LIN {X 0,Y 517.926,Z 485.108,A -85,B 0,C 180,E1 -5117.361,E2 -5117.361} C_VEL
LIN {X 0,Y 517.662,Z 497.086,A -85,B 0,C 180,E1 -5118.063,E2 -5118.063} C_VEL
LIN {X 0,Y 517.369,Z 508.755,A -85,B 0,C 180,E1 -5118.938,E2 -5118.938} C_VEL
LIN {X 0,Y 517.043,Z 518.274,A -85,B 0,C 180,E1 -5119.822,E2 -5119.822} C_VEL
LIN {X 0,Y 516.815,Z 526.96,A -85,B 0,C 180,E1 -5120.806,E2 -5120.806} C_VEL
LIN {X 0,Y 516.617,Z 535.392,A -85,B 0,C 180,E1 -5121.985,E2 -5121.985} C_VEL
LIN {X 0,Y 516.477,Z 542.404,A -85,B 0,C 180,E1 -5123.204,E2 -5123.204} C_VEL
LIN {X 0,Y 516.405,Z 548.407,A -85,B 0,C 180,E1 -5124.533,E2 -5124.533} C_VEL
LIN {X 0,Y 516.343,Z 552.44,A -85,B 0,C 180,E1 -5125.707,E2 -5125.707} C_VEL
LIN {X 0,Y 516.282,Z 555.413,A -85,B 0,C 180,E1 -5126.879,E2 -5126.879} C_VEL
LIN {X 0,Y 516.261,Z 556.832,A -85,B 0,C 180,E1 -5127.659,E2 -5127.659} C_VEL
LIN {X 0,Y 516.16,Z 558.451,A -85,B 0,C 180,E1 -5129.22,E2 -5129.22} C_VEL
LIN {X 0,Y 516.155,Z 558.67,A -85,B 0,C 180,E1 -5130,E2 -5130} C_VEL
LIN {X 0,Y 516.16,Z 558.45,A -85,B 0,C 180,E1 -5130.78,E2 -5130.78} C_VEL
LIN {X 0,Y 516.261,Z 556.828,A -85,B 0,C 180,E1 -5132.341,E2 -5132.341} C_VEL
LIN {X 0,Y 516.282,Z 555.406,A -85,B 0,C 180,E1 -5133.121,E2 -5133.121} C_VEL
LIN {X 0,Y 516.343,Z 552.421,A -85,B 0,C 180,E1 -5134.293,E2 -5134.293} C_VEL
LIN {X 0,Y 516.405,Z 548.374,A -85,B 0,C 180,E1 -5135.467,E2 -5135.467} C_VEL
LIN {X 0,Y 516.465,Z 542.972,A -85,B 0,C 180,E1 -5136.679,E2 -5136.679} C_VEL
LIN {X 0,Y 516.579,Z 536.576,A -85,B 0,C 180,E1 -5137.819,E2 -5137.819} C_VEL
LIN {X 0,Y 516.771,Z 528.376,A -85,B 0,C 180,E1 -5138.998,E2 -5138.998} C_VEL
LIN {X 0,Y 516.993,Z 520.003,A -85,B 0,C 180,E1 -5139.981,E2 -5139.981} C_VEL
LIN {X 0,Y 517.292,Z 509.755,A -85,B 0,C 180,E1 -5140.965,E2 -5140.965} C_VEL
LIN {X 0,Y 517.549,Z 499.569,A -85,B 0,C 180,E1 -5141.753,E2 -5141.753} C_VEL
LIN {X 0,Y 517.84,Z 487.976,A -85,B 0,C 180,E1 -5142.47,E2 -5142.47} C_VEL
LIN {X 0,Y 518.063,Z 476.175,A -85,B 0,C 180,E1 -5143.034,E2 -5143.034} C_VEL
LIN {X 0,Y 518.291,Z 463.332,A -85,B 0,C 180,E1 -5143.478,E2 -5143.478} C_VEL
LIN {X 0,Y 518.127,Z 456.266,A -85,B 0,C 180,E1 -5143.657,E2 -5143.657} C_VEL
LIN {X 0,Y 516.991,Z 447.207,A -85,B 0,C 180,E1 -5143.863,E2 -5143.863} C_VEL
LIN {X 0,Y 517.273,Z 430.127,A -85,B 0,C 180,E1 -5146.781,E2 -5146.781} C_VEL
LIN {X 0,Y 517.596,Z 415.01,A -85,B 0,C 180,E1 -5149.431,E2 -5149.431} C_VEL
LIN {X 0,Y 517.925,Z 402.35,A -85,B 0,C 180,E1 -5151.702,E2 -5151.702} C_VEL
LIN {X 0,Y 518.488,Z 388.132,A -85,B 0,C 180,E1 -5154.383,E2 -5154.383} C_VEL
LIN {X 0,Y 519.352,Z 373.06,A -85,B 0,C 180,E1 -5157.394,E2 -5157.394} C_VEL
LIN {X 0,Y 519.545,Z 368.168,A -85,B 0,C 180,E1 -5158.445,E2 -5158.445} C_VEL
LIN {X 0,Y 517.68,Z 359.516,A -85,B 0,C 180,E1 -5160.604,E2 -5160.604} C_VEL
LIN {X 0,Y 516.886,Z 356.103,A -85,B 0,C 180,E1 -5161.566,E2 -5161.566} C_VEL
LIN {X 0,Y 516.911,Z 356.099,A -85,B 0,C 180,E1 -5163.966,E2 -5163.966} C_VEL
LIN {X 0,Y 516.879,Z 356.103,A -85,B 0,C 180,E1 -5166.746,E2 -5166.746} C_VEL
LIN {X 0,Y 516.885,Z 356.102,A -85,B 0,C 180,E1 -5169.721,E2 -5169.721} C_VEL
LIN {X 0,Y 516.91,Z 356.1,A -85,B 0,C 180,E1 -5172.761,E2 -5172.761} C_VEL
LIN {X 0,Y 516.926,Z 356.097,A -85,B 0,C 180,E1 -5175.01,E2 -5175.01} C_VEL
LIN {X 0,Y 516.921,Z 356.097,A -85,B 0,C 180,E1 -5178.398,E2 -5178.398} C_VEL
LIN {X 0,Y 516.91,Z 356.1,A -85,B 0,C 180,E1 -5181.287,E2 -5181.287} C_VEL
LIN {X 0,Y 516.89,Z 356.103,A -85,B 0,C 180,E1 -5184.221,E2 -5184.221} C_VEL
LIN {X 0,Y 516.9,Z 356.102,A -85,B 0,C 180,E1 -5187.053,E2 -5187.053} C_VEL
LIN {X 0,Y 516.926,Z 356.236,A -85,B 0,C 180,E1 -5189.153,E2 -5189.153} C_VEL
LIN {X 0,Y 517.195,Z 359.452,A -85,B 0,C 180,E1 -5190.712,E2 -5190.712} C_VEL
LIN {X 0,Y 517.047,Z 365.951,A -85,B 0,C 180,E1 -5193.781,E2 -5193.781} C_VEL
LIN {X 0,Y 516.896,Z 372.331,A -85,B 0,C 180,E1 -5196.778,E2 -5196.778} C_VEL
LIN {X 0,Y 516.762,Z 378.758,A -85,B 0,C 180,E1 -5199.786,E2 -5199.786} C_VEL
LIN {X 0,Y 516.703,Z 384.815,A -85,B 0,C 180,E1 -5202.588,E2 -5202.588} C_VEL
LIN {X 0,Y 516.634,Z 390.136,A -85,B 0,C 180,E1 -5205.021,E2 -5205.021} C_VEL
LIN {X 0,Y 516.491,Z 397.626,A -85,B 0,C 180,E1 -5208.442,E2 -5208.442} C_VEL
LIN {X 0,Y 516.412,Z 405.171,A -85,B 0,C 180,E1 -5211.809,E2 -5211.809} C_VEL
LIN {X 0,Y 517.193,Z 411.851,A -85,B 0,C 180,E1 -5212.092,E2 -5212.092} C_VEL
LIN {X 0,Y 517.076,Z 421.865,A -85,B 0,C 180,E1 -5212.62,E2 -5212.62} C_VEL
LIN {X 0,Y 516.967,Z 430.533,A -85,B 0,C 180,E1 -5213.252,E2 -5213.252} C_VEL
LIN {X 0,Y 516.779,Z 437.867,A -85,B 0,C 180,E1 -5213.95,E2 -5213.95} C_VEL
LIN {X 0,Y 516.671,Z 444.225,A -85,B 0,C 180,E1 -5214.732,E2 -5214.732} C_VEL
LIN {X 0,Y 516.564,Z 449.253,A -85,B 0,C 180,E1 -5215.513,E2 -5215.513} C_VEL
LIN {X 0,Y 516.546,Z 454.014,A -85,B 0,C 180,E1 -5216.49,E2 -5216.49} C_VEL
LIN {X 0,Y 516.333,Z 457.969,A -85,B 0,C 180,E1 -5217.66,E2 -5217.66} C_VEL
LIN {X 0,Y 516.266,Z 459.663,A -85,B 0,C 180,E1 -5218.44,E2 -5218.44} C_VEL
LIN {X 0,Y 516.246,Z 460.666,A -85,B 0,C 180,E1 -5219.22,E2 -5219.22} C_VEL
LIN {X 0,Y 516.24,Z 461.005,A -85,B 0,C 180,E1 -5220,E2 -5220} C_VEL
LIN {X 0,Y 516.239,Z 460.689,A -85,B 0,C 180,E1 -5220.78,E2 -5220.78} C_VEL
LIN {X 0,Y 516.255,Z 459.71,A -85,B 0,C 180,E1 -5221.56,E2 -5221.56} C_VEL
LIN {X 0,Y 516.421,Z 456.909,A -85,B 0,C 180,E1 -5222.73,E2 -5222.73} C_VEL
LIN {X 0,Y 516.543,Z 454.125,A -85,B 0,C 180,E1 -5223.51,E2 -5223.51} C_VEL
LIN {X 0,Y 516.558,Z 449.409,A -85,B 0,C 180,E1 -5224.487,E2 -5224.487} C_VEL
LIN {X 0,Y 516.634,Z 444.423,A -85,B 0,C 180,E1 -5225.269,E2 -5225.269} C_VEL
LIN {X 0,Y 516.662,Z 438.145,A -85,B 0,C 180,E1 -5226.052,E2 -5226.052} C_VEL
LIN {X 0,Y 516.878,Z 430.436,A -85,B 0,C 180,E1 -5226.788,E2 -5226.788} C_VEL
LIN {X 0,Y 516.993,Z 421.754,A -85,B 0,C 180,E1 -5227.42,E2 -5227.42} C_VEL
LIN {X 0,Y 517.128,Z 411.453,A -85,B 0,C 180,E1 -5227.958,E2 -5227.958} C_VEL
LIN {X 0,Y 516.329,Z 404.462,A -85,B 0,C 180,E1 -5228.242,E2 -5228.242} C_VEL
LIN {X 0,Y 516.353,Z 396.845,A -85,B 0,C 180,E1 -5231.483,E2 -5231.483} C_VEL
LIN {X 0,Y 516.469,Z 389.182,A -85,B 0,C 180,E1 -5234.949,E2 -5234.949} C_VEL
LIN {X 0,Y 516.579,Z 382.087,A -85,B 0,C 180,E1 -5238.235,E2 -5238.235} C_VEL
LIN {X 0,Y 516.645,Z 376.784,A -85,B 0,C 180,E1 -5240.713,E2 -5240.713} C_VEL
LIN {X 0,Y 516.693,Z 371.107,A -85,B 0,C 180,E1 -5243.232,E2 -5243.232} C_VEL
LIN {X 0,Y 516.825,Z 364.647,A -85,B 0,C 180,E1 -5246.169,E2 -5246.169} C_VEL
LIN {X 0,Y 516.974,Z 357.423,A -85,B 0,C 180,E1 -5249.535,E2 -5249.535} C_VEL
LIN {X 0,Y 517.006,Z 356.086,A -85,B 0,C 180,E1 -5250.197,E2 -5250.197} C_VEL
LIN {X 0,Y 516.915,Z 356.093,A -85,B 0,C 180,E1 -5253.879,E2 -5253.879} C_VEL
LIN {X 0,Y 516.886,Z 356.099,A -85,B 0,C 180,E1 -5256.746,E2 -5256.746} C_VEL
LIN {X 0,Y 516.886,Z 356.101,A -85,B 0,C 180,E1 -5259.721,E2 -5259.721} C_VEL
LIN {X 0,Y 516.917,Z 356.095,A -85,B 0,C 180,E1 -5261.775,E2 -5261.775} C_VEL
LIN {X 0,Y 516.927,Z 356.094,A -85,B 0,C 180,E1 -5265.01,E2 -5265.01} C_VEL
LIN {X 0,Y 516.92,Z 356.095,A -85,B 0,C 180,E1 -5268.398,E2 -5268.398} C_VEL
LIN {X 0,Y 516.886,Z 356.101,A -85,B 0,C 180,E1 -5269.481,E2 -5269.481} C_VEL
LIN {X 0,Y 516.226,Z 356.185,A -85,B 0,C 180,E1 -5270.132,E2 -5270.132} C_VEL
LIN {X 0,Y 513.357,Z 356.543,A -85,B 0,C 180,E1 -5271.189,E2 -5271.189} C_VEL
LIN {X 0,Y 510.931,Z 356.843,A -85,B 0,C 180,E1 -5272.04,E2 -5272.04} C_VEL
LIN {X 0,Y 509.898,Z 356.972,A -85,B 0,C 180,E1 -5272.697,E2 -5272.697} C_VEL
LIN {X 0,Y 509.818,Z 356.981,A -85,B 0,C 180,E1 -5272.92,E2 -5272.92} C_VEL
LIN {X 0,Y 509.86,Z 356.973,A -85,B 0,C 180,E1 -5275.797,E2 -5275.797} C_VEL
LIN {X 0,Y 509.85,Z 356.975,A -85,B 0,C 180,E1 -5278.72,E2 -5278.72} C_VEL
LIN {X 0,Y 509.902,Z 356.969,A -85,B 0,C 180,E1 -5281.899,E2 -5281.899} C_VEL
LIN {X 0,Y 509.845,Z 356.979,A -85,B 0,C 180,E1 -5284.702,E2 -5284.702} C_VEL
LIN {X 0,Y 509.831,Z 356.977,A -85,B 0,C 180,E1 -5287.458,E2 -5287.458} C_VEL
LIN {X 0,Y 509.921,Z 356.97,A -85,B 0,C 180,E1 -5289.845,E2 -5289.845} C_VEL
LIN {X 0,Y 509.886,Z 356.973,A -85,B 0,C 180,E1 -5293.175,E2 -5293.175} C_VEL
LIN {X 0,Y 509.868,Z 356.972,A -85,B 0,C 180,E1 -5295.634,E2 -5295.634} C_VEL
LIN {X 0,Y 509.918,Z 356.966,A -85,B 0,C 180,E1 -5298.875,E2 -5298.875} C_VEL
LIN {X 0,Y 509.956,Z 356.962,A -85,B 0,C 180,E1 -5302.078,E2 -5302.078} C_VEL
LIN {X 0,Y 509.985,Z 356.962,A -85,B 0,C 180,E1 -5304.464,E2 -5304.464} C_VEL
LIN {X 0,Y 510.059,Z 356.949,A -85,B 0,C 180,E1 -5307.631,E2 -5307.631} C_VEL
LIN {X 0,Y 510.068,Z 356.948,A -85,B 0,C 180,E1 -5310.789,E2 -5310.789} C_VEL
LIN {X 0,Y 509.958,Z 356.965,A -85,B 0,C 180,E1 -5313.16,E2 -5313.16} C_VEL
LIN {X 0,Y 509.958,Z 356.965,A -85,B 0,C 180,E1 -5316.33,E2 -5316.33} C_VEL
LIN {X 0,Y 509.919,Z 356.964,A -85,B 0,C 180,E1 -5318.72,E2 -5318.72} C_VEL
LIN {X 0,Y 509.909,Z 356.968,A -85,B 0,C 180,E1 -5321.932,E2 -5321.932} C_VEL
LIN {X 0,Y 509.898,Z 356.969,A -85,B 0,C 180,E1 -5325.242,E2 -5325.242} C_VEL
LIN {X 0,Y 509.893,Z 356.974,A -85,B 0,C 180,E1 -5328.001,E2 -5328.001} C_VEL
LIN {X 0,Y 509.854,Z 356.975,A -85,B 0,C 180,E1 -5331.002,E2 -5331.002} C_VEL
LIN {X 0,Y 509.869,Z 356.975,A -85,B 0,C 180,E1 -5334.426,E2 -5334.426} C_VEL
LIN {X 0,Y 509.889,Z 356.97,A -85,B 0,C 180,E1 -5337.055,E2 -5337.055} C_VEL
LIN {X 0,Y 509.861,Z 356.977,A -85,B 0,C 180,E1 -5339.751,E2 -5339.751} C_VEL
LIN {X 0,Y 509.878,Z 356.973,A -85,B 0,C 180,E1 -5342.774,E2 -5342.774} C_VEL
LIN {X 0,Y 509.829,Z 356.977,A -85,B 0,C 180,E1 -5345.578,E2 -5345.578} C_VEL
LIN {X 0,Y 509.854,Z 356.977,A -85,B 0,C 180,E1 -5348.338,E2 -5348.338} C_VEL
LIN {X 0,Y 509.858,Z 356.978,A -85,B 0,C 180,E1 -5351.425,E2 -5351.425} C_VEL
LIN {X 0,Y 509.86,Z 356.977,A -85,B 0,C 180,E1 -5354.668,E2 -5354.668} C_VEL
LIN {X 0,Y 509.858,Z 356.977,A -85,B 0,C 180,E1 -5358.103,E2 -5358.103} C_VEL
LIN {X 0,Y 509.849,Z 356.974,A -85,B 0,C 180,E1 -5360.647,E2 -5360.647} C_VEL
LIN {X 0,Y 509.827,Z 356.977,A -85,B 0,C 180,E1 -5363.647,E2 -5363.647} C_VEL
LIN {X 0,Y 509.862,Z 356.978,A -85,B 0,C 180,E1 -5366.539,E2 -5366.539} C_VEL
LIN {X 0,Y 509.848,Z 356.977,A -85,B 0,C 180,E1 -5369.334,E2 -5369.334} C_VEL
LIN {X 0,Y 509.895,Z 356.968,A -85,B 0,C 180,E1 -5372.054,E2 -5372.054} C_VEL
LIN {X 0,Y 509.88,Z 356.975,A -85,B 0,C 180,E1 -5374.704,E2 -5374.704} C_VEL
LIN {X 0,Y 509.84,Z 356.976,A -85,B 0,C 180,E1 -5377.455,E2 -5377.455} C_VEL
LIN {X 0,Y 509.92,Z 356.969,A -85,B 0,C 180,E1 -5379.845,E2 -5379.845} C_VEL
LIN {X 0,Y 509.887,Z 356.973,A -85,B 0,C 180,E1 -5383.175,E2 -5383.175} C_VEL
LIN {X 0,Y 509.867,Z 356.971,A -85,B 0,C 180,E1 -5385.634,E2 -5385.634} C_VEL
LIN {X 0,Y 509.925,Z 356.965,A -85,B 0,C 180,E1 -5388.875,E2 -5388.875} C_VEL
LIN {X 0,Y 509.955,Z 356.962,A -85,B 0,C 180,E1 -5392.078,E2 -5392.078} C_VEL
LIN {X 0,Y 509.985,Z 356.96,A -85,B 0,C 180,E1 -5394.464,E2 -5394.464} C_VEL
LIN {X 0,Y 510.058,Z 356.949,A -85,B 0,C 180,E1 -5397.631,E2 -5397.631} C_VEL
LIN {X 0,Y 510.067,Z 356.948,A -85,B 0,C 180,E1 -5400.789,E2 -5400.789} C_VEL
LIN {X 0,Y 509.96,Z 356.964,A -85,B 0,C 180,E1 -5403.16,E2 -5403.16} C_VEL
LIN {X 0,Y 509.981,Z 356.962,A -85,B 0,C 180,E1 -5406.33,E2 -5406.33} C_VEL
LIN {X 0,Y 509.915,Z 356.967,A -85,B 0,C 180,E1 -5408.72,E2 -5408.72} C_VEL
LIN {X 0,Y 509.907,Z 356.969,A -85,B 0,C 180,E1 -5411.932,E2 -5411.932} C_VEL
LIN {X 0,Y 509.897,Z 356.97,A -85,B 0,C 180,E1 -5415.242,E2 -5415.242} C_VEL
LIN {X 0,Y 509.869,Z 356.975,A -85,B 0,C 180,E1 -5417.993,E2 -5417.993} C_VEL
LIN {X 0,Y 509.889,Z 356.97,A -85,B 0,C 180,E1 -5420.402,E2 -5420.402} C_VEL
LIN {X 0,Y 509.832,Z 356.979,A -85,B 0,C 180,E1 -5423.563,E2 -5423.563} C_VEL
LIN {X 0,Y 509.914,Z 356.972,A -85,B 0,C 180,E1 -5426.378,E2 -5426.378} C_VEL
LIN {X 0,Y 509.879,Z 356.969,A -85,B 0,C 180,E1 -5428.844,E2 -5428.844} C_VEL
LIN {X 0,Y 509.823,Z 356.983,A -85,B 0,C 180,E1 -5431.59,E2 -5431.59} C_VEL
LIN {X 0,Y 509.855,Z 356.976,A -85,B 0,C 180,E1 -5434.413,E2 -5434.413} C_VEL
LIN {X 0,Y 509.822,Z 356.978,A -85,B 0,C 180,E1 -5437.34,E2 -5437.34} C_VEL
LIN {X 0,Y 509.84,Z 356.975,A -85,B 0,C 180,E1 -5440.382,E2 -5440.382} C_VEL
LIN {X 0,Y 509.842,Z 356.979,A -85,B 0,C 180,E1 -5443.064,E2 -5443.064} C_VEL
LIN {X 0,Y 509.833,Z 356.977,A -85,B 0,C 180,E1 -5445.792,E2 -5445.792} C_VEL
LIN {X 0,Y 509.86,Z 356.974,A -85,B 0,C 180,E1 -5448.575,E2 -5448.575} C_VEL
LIN {X 0,Y 509.853,Z 356.976,A -85,B 0,C 180,E1 -5451.787,E2 -5451.787} C_VEL
LIN {X 0,Y 509.832,Z 356.981,A -85,B 0,C 180,E1 -5454.622,E2 -5454.622} C_VEL
LIN {X 0,Y 509.866,Z 356.97,A -85,B 0,C 180,E1 -5457.481,E2 -5457.481} C_VEL
LIN {X 0,Y 509.875,Z 357.124,A -85,B 0,C 180,E1 -5458.865,E2 -5458.865} C_VEL
LIN {X 0,Y 512.351,Z 368.579,A -85,B 0,C 180,E1 -5461.39,E2 -5461.39} C_VEL
LIN {X 0,Y 512.386,Z 374.915,A -85,B 0,C 180,E1 -5462.646,E2 -5462.646} C_VEL
LIN {X 0,Y 511.54,Z 391.643,A -85,B 0,C 180,E1 -5465.875,E2 -5465.875} C_VEL
LIN {X 0,Y 510.912,Z 408.335,A -85,B 0,C 180,E1 -5469.044,E2 -5469.044} C_VEL
LIN {X 0,Y 510.492,Z 420.904,A -85,B 0,C 180,E1 -5471.332,E2 -5471.332} C_VEL
LIN {X 0,Y 510.154,Z 437.346,A -85,B 0,C 180,E1 -5474.204,E2 -5474.204} C_VEL
LIN {X 0,Y 509.97,Z 447.553,A -85,B 0,C 180,E1 -5475.994,E2 -5475.994} C_VEL
LIN {X 0,Y 511.367,Z 459.455,A -85,B 0,C 180,E1 -5476.261,E2 -5476.261} C_VEL
LIN {X 0,Y 511.148,Z 472.764,A -85,B 0,C 180,E1 -5476.685,E2 -5476.685} C_VEL
LIN {X 0,Y 510.938,Z 483.958,A -85,B 0,C 180,E1 -5477.185,E2 -5477.185} C_VEL
LIN {X 0,Y 510.66,Z 495.859,A -85,B 0,C 180,E1 -5477.878,E2 -5477.878} C_VEL
LIN {X 0,Y 510.293,Z 507.862,A -85,B 0,C 180,E1 -5478.782,E2 -5478.782} C_VEL
LIN {X 0,Y 510.011,Z 517.448,A -85,B 0,C 180,E1 -5479.68,E2 -5479.68} C_VEL
LIN {X 0,Y 509.759,Z 526.189,A -85,B 0,C 180,E1 -5480.677,E2 -5480.677} C_VEL
LIN {X 0,Y 509.538,Z 534.661,A -85,B 0,C 180,E1 -5481.872,E2 -5481.872} C_VEL
LIN {X 0,Y 509.401,Z 541.938,A -85,B 0,C 180,E1 -5483.156,E2 -5483.156} C_VEL
LIN {X 0,Y 509.344,Z 547.728,A -85,B 0,C 180,E1 -5484.457,E2 -5484.457} C_VEL
LIN {X 0,Y 509.268,Z 551.771,A -85,B 0,C 180,E1 -5485.647,E2 -5485.647} C_VEL
LIN {X 0,Y 509.232,Z 554.754,A -85,B 0,C 180,E1 -5486.835,E2 -5486.835} C_VEL
LIN {X 0,Y 509.19,Z 556.176,A -85,B 0,C 180,E1 -5487.627,E2 -5487.627} C_VEL
LIN {X 0,Y 509.09,Z 557.796,A -85,B 0,C 180,E1 -5489.209,E2 -5489.209} C_VEL
LIN {X 0,Y 509.086,Z 558.01,A -85,B 0,C 180,E1 -5490,E2 -5490} C_VEL
LIN {X 0,Y 509.09,Z 557.787,A -85,B 0,C 180,E1 -5490.791,E2 -5490.791} C_VEL
LIN {X 0,Y 509.19,Z 556.154,A -85,B 0,C 180,E1 -5492.373,E2 -5492.373} C_VEL
LIN {X 0,Y 509.232,Z 554.722,A -85,B 0,C 180,E1 -5493.165,E2 -5493.165} C_VEL
LIN {X 0,Y 509.268,Z 551.718,A -85,B 0,C 180,E1 -5494.353,E2 -5494.353} C_VEL
LIN {X 0,Y 509.344,Z 547.65,A -85,B 0,C 180,E1 -5495.543,E2 -5495.543} C_VEL
LIN {X 0,Y 509.402,Z 541.835,A -85,B 0,C 180,E1 -5496.844,E2 -5496.844} C_VEL
LIN {X 0,Y 509.563,Z 534.524,A -85,B 0,C 180,E1 -5498.127,E2 -5498.127} C_VEL
LIN {X 0,Y 509.759,Z 526.001,A -85,B 0,C 180,E1 -5499.323,E2 -5499.323} C_VEL
LIN {X 0,Y 510.006,Z 517.207,A -85,B 0,C 180,E1 -5500.32,E2 -5500.32} C_VEL
LIN {X 0,Y 510.33,Z 506.364,A -85,B 0,C 180,E1 -5501.317,E2 -5501.317} C_VEL
LIN {X 0,Y 510.599,Z 495.788,A -85,B 0,C 180,E1 -5502.101,E2 -5502.101} C_VEL
LIN {X 0,Y 510.848,Z 485.428,A -85,B 0,C 180,E1 -5502.716,E2 -5502.716} C_VEL
LIN {X 0,Y 511.114,Z 473.406,A -85,B 0,C 180,E1 -5503.265,E2 -5503.265} C_VEL
LIN {X 0,Y 511.354,Z 460.421,A -85,B 0,C 180,E1 -5503.689,E2 -5503.689} C_VEL
LIN {X 0,Y 510.48,Z 452.043,A -85,B 0,C 180,E1 -5503.897,E2 -5503.897} C_VEL
LIN {X 0,Y 509.898,Z 446.891,A -85,B 0,C 180,E1 -5504.009,E2 -5504.009} C_VEL
LIN {X 0,Y 510.228,Z 430.816,A -85,B 0,C 180,E1 -5506.814,E2 -5506.814} C_VEL
LIN {X 0,Y 510.643,Z 413.461,A -85,B 0,C 180,E1 -5509.916,E2 -5509.916} C_VEL
LIN {X 0,Y 511.166,Z 398.782,A -85,B 0,C 180,E1 -5512.642,E2 -5512.642} C_VEL
LIN {X 0,Y 511.803,Z 384.679,A -85,B 0,C 180,E1 -5515.412,E2 -5515.412} C_VEL
LIN {X 0,Y 512.602,Z 373.258,A -85,B 0,C 180,E1 -5517.785,E2 -5517.785} C_VEL
LIN {X 0,Y 512.57,Z 369.319,A -85,B 0,C 180,E1 -5518.679,E2 -5518.679} C_VEL
LIN {X 0,Y 510.99,Z 361.886,A -85,B 0,C 180,E1 -5520.59,E2 -5520.59} C_VEL
LIN {X 0,Y 509.837,Z 356.98,A -85,B 0,C 180,E1 -5521.996,E2 -5521.996} C_VEL
LIN {X 0,Y 509.85,Z 356.979,A -85,B 0,C 180,E1 -5524.414,E2 -5524.414} C_VEL
LIN {X 0,Y 509.819,Z 356.984,A -85,B 0,C 180,E1 -5527.341,E2 -5527.341} C_VEL
LIN {X 0,Y 509.841,Z 356.98,A -85,B 0,C 180,E1 -5530.382,E2 -5530.382} C_VEL
LIN {X 0,Y 509.843,Z 356.979,A -85,B 0,C 180,E1 -5533.064,E2 -5533.064} C_VEL
LIN {X 0,Y 509.834,Z 356.981,A -85,B 0,C 180,E1 -5535.792,E2 -5535.792} C_VEL
LIN {X 0,Y 509.864,Z 356.976,A -85,B 0,C 180,E1 -5538.575,E2 -5538.575} C_VEL
LIN {X 0,Y 509.859,Z 356.978,A -85,B 0,C 180,E1 -5541.786,E2 -5541.786} C_VEL
LIN {X 0,Y 509.846,Z 356.979,A -85,B 0,C 180,E1 -5544.623,E2 -5544.623} C_VEL
LIN {X 0,Y 509.866,Z 356.978,A -85,B 0,C 180,E1 -5547.481,E2 -5547.481} C_VEL
LIN {X 0,Y 509.878,Z 357.064,A -85,B 0,C 180,E1 -5548.865,E2 -5548.865} C_VEL
LIN {X 0,Y 510.185,Z 359.87,A -85,B 0,C 180,E1 -5550.27,E2 -5550.27} C_VEL
LIN {X 0,Y 510.046,Z 366.764,A -85,B 0,C 180,E1 -5553.592,E2 -5553.592} C_VEL
LIN {X 0,Y 509.892,Z 372.726,A -85,B 0,C 180,E1 -5556.44,E2 -5556.44} C_VEL
LIN {X 0,Y 509.764,Z 379.479,A -85,B 0,C 180,E1 -5559.637,E2 -5559.637} C_VEL
LIN {X 0,Y 509.676,Z 385.234,A -85,B 0,C 180,E1 -5562.34,E2 -5562.34} C_VEL
LIN {X 0,Y 509.499,Z 392.365,A -85,B 0,C 180,E1 -5565.624,E2 -5565.624} C_VEL
LIN {X 0,Y 509.441,Z 399.439,A -85,B 0,C 180,E1 -5568.864,E2 -5568.864} C_VEL
LIN {X 0,Y 509.374,Z 405.65,A -85,B 0,C 180,E1 -5571.67,E2 -5571.67} C_VEL
LIN {X 0,Y 510.197,Z 411.929,A -85,B 0,C 180,E1 -5571.933,E2 -5571.933} C_VEL
LIN {X 0,Y 510.145,Z 421.091,A -85,B 0,C 180,E1 -5572.41,E2 -5572.41} C_VEL
LIN {X 0,Y 509.995,Z 429.686,A -85,B 0,C 180,E1 -5573.02,E2 -5573.02} C_VEL
LIN {X 0,Y 509.821,Z 436.773,A -85,B 0,C 180,E1 -5573.668,E2 -5573.668} C_VEL
LIN {X 0,Y 509.618,Z 443.544,A -85,B 0,C 180,E1 -5574.46,E2 -5574.46} C_VEL
LIN {X 0,Y 509.541,Z 448.832,A -85,B 0,C 180,E1 -5575.253,E2 -5575.253} C_VEL
LIN {X 0,Y 509.471,Z 453.003,A -85,B 0,C 180,E1 -5576.045,E2 -5576.045} C_VEL
LIN {X 0,Y 509.392,Z 456.24,A -85,B 0,C 180,E1 -5576.836,E2 -5576.836} C_VEL
LIN {X 0,Y 509.274,Z 458.669,A -85,B 0,C 180,E1 -5577.627,E2 -5577.627} C_VEL
LIN {X 0,Y 509.204,Z 460.357,A -85,B 0,C 180,E1 -5578.418,E2 -5578.418} C_VEL
LIN {X 0,Y 509.181,Z 461.352,A -85,B 0,C 180,E1 -5579.209,E2 -5579.209} C_VEL
LIN {X 0,Y 509.173,Z 461.683,A -85,B 0,C 180,E1 -5580,E2 -5580} C_VEL
LIN {X 0,Y 509.172,Z 461.357,A -85,B 0,C 180,E1 -5580.791,E2 -5580.791} C_VEL
LIN {X 0,Y 509.189,Z 460.367,A -85,B 0,C 180,E1 -5581.582,E2 -5581.582} C_VEL
LIN {X 0,Y 509.378,Z 457.553,A -85,B 0,C 180,E1 -5582.768,E2 -5582.768} C_VEL
LIN {X 0,Y 509.51,Z 454.754,A -85,B 0,C 180,E1 -5583.559,E2 -5583.559} C_VEL
LIN {X 0,Y 509.524,Z 450.019,A -85,B 0,C 180,E1 -5584.549,E2 -5584.549} C_VEL
LIN {X 0,Y 509.592,Z 445.031,A -85,B 0,C 180,E1 -5585.342,E2 -5585.342} C_VEL
LIN {X 0,Y 509.628,Z 438.744,A -85,B 0,C 180,E1 -5586.135,E2 -5586.135} C_VEL
LIN {X 0,Y 509.889,Z 430.44,A -85,B 0,C 180,E1 -5586.933,E2 -5586.933} C_VEL
LIN {X 0,Y 510.004,Z 422.417,A -85,B 0,C 180,E1 -5587.522,E2 -5587.522} C_VEL
LIN {X 0,Y 510.154,Z 412.291,A -85,B 0,C 180,E1 -5588.068,E2 -5588.068} C_VEL
LIN {X 0,Y 509.285,Z 404.753,A -85,B 0,C 180,E1 -5588.381,E2 -5588.381} C_VEL
LIN {X 0,Y 509.289,Z 397.433,A -85,B 0,C 180,E1 -5591.542,E2 -5591.542} C_VEL
LIN {X 0,Y 509.362,Z 391.043,A -85,B 0,C 180,E1 -5594.38,E2 -5594.38} C_VEL
LIN {X 0,Y 509.485,Z 384.018,A -85,B 0,C 180,E1 -5597.667,E2 -5597.667} C_VEL
LIN {X 0,Y 509.568,Z 378.373,A -85,B 0,C 180,E1 -5600.304,E2 -5600.304} C_VEL
LIN {X 0,Y 509.637,Z 372.997,A -85,B 0,C 180,E1 -5602.714,E2 -5602.714} C_VEL
LIN {X 0,Y 509.749,Z 367.417,A -85,B 0,C 180,E1 -5605.303,E2 -5605.303} C_VEL
LIN {X 0,Y 509.851,Z 361.435,A -85,B 0,C 180,E1 -5608.09,E2 -5608.09} C_VEL
LIN {X 0,Y 509.966,Z 356.963,A -85,B 0,C 180,E1 -5610.257,E2 -5610.257} C_VEL
LIN {X 0,Y 509.865,Z 356.972,A -85,B 0,C 180,E1 -5613.461,E2 -5613.461} C_VEL
LIN {X 0,Y 509.838,Z 356.98,A -85,B 0,C 180,E1 -5616.352,E2 -5616.352} C_VEL
LIN {X 0,Y 509.839,Z 356.98,A -85,B 0,C 180,E1 -5619.471,E2 -5619.471} C_VEL
LIN {X 0,Y 509.837,Z 356.977,A -85,B 0,C 180,E1 -5622.49,E2 -5622.49} C_VEL
LIN {X 0,Y 509.861,Z 356.973,A -85,B 0,C 180,E1 -5625.332,E2 -5625.332} C_VEL
LIN {X 0,Y 509.861,Z 356.974,A -85,B 0,C 180,E1 -5628.575,E2 -5628.575} C_VEL
LIN {X 0,Y 509.854,Z 356.975,A -85,B 0,C 180,E1 -5631.787,E2 -5631.787} C_VEL
LIN {X 0,Y 509.818,Z 356.981,A -85,B 0,C 180,E1 -5632.92,E2 -5632.92} C_VEL
LIN {X 0,Y 509.164,Z 357.064,A -85,B 0,C 180,E1 -5633.58,E2 -5633.58} C_VEL
LIN {X 0,Y 506.315,Z 357.42,A -85,B 0,C 180,E1 -5634.651,E2 -5634.651} C_VEL
LIN {X 0,Y 503.905,Z 357.717,A -85,B 0,C 180,E1 -5635.514,E2 -5635.514} C_VEL
LIN {X 0,Y 502.88,Z 357.846,A -85,B 0,C 180,E1 -5636.18,E2 -5636.18} C_VEL
LIN {X 0,Y 502.802,Z 357.851,A -85,B 0,C 180,E1 -5636.406,E2 -5636.406} C_VEL
LIN {X 0,Y 502.813,Z 357.855,A -85,B 0,C 180,E1 -5639.789,E2 -5639.789} C_VEL
LIN {X 0,Y 502.838,Z 357.85,A -85,B 0,C 180,E1 -5642.533,E2 -5642.533} C_VEL
LIN {X 0,Y 502.807,Z 357.85,A -85,B 0,C 180,E1 -5645.305,E2 -5645.305} C_VEL
LIN {X 0,Y 502.784,Z 357.857,A -85,B 0,C 180,E1 -5647.826,E2 -5647.826} C_VEL
LIN {X 0,Y 502.828,Z 357.85,A -85,B 0,C 180,E1 -5650.4,E2 -5650.4} C_VEL
LIN {X 0,Y 502.834,Z 357.852,A -85,B 0,C 180,E1 -5652.932,E2 -5652.932} C_VEL
LIN {X 0,Y 502.849,Z 357.846,A -85,B 0,C 180,E1 -5655.429,E2 -5655.429} C_VEL
LIN {X 0,Y 502.882,Z 357.842,A -85,B 0,C 180,E1 -5658.717,E2 -5658.717} C_VEL
LIN {X 0,Y 502.906,Z 357.84,A -85,B 0,C 180,E1 -5661.967,E2 -5661.967} C_VEL
LIN {X 0,Y 502.938,Z 357.839,A -85,B 0,C 180,E1 -5664.386,E2 -5664.386} C_VEL
LIN {X 0,Y 503.029,Z 357.825,A -85,B 0,C 180,E1 -5667.598,E2 -5667.598} C_VEL
LIN {X 0,Y 503.032,Z 357.826,A -85,B 0,C 180,E1 -5670,E2 -5670} C_VEL
LIN {X 0,Y 503.029,Z 357.825,A -85,B 0,C 180,E1 -5672.402,E2 -5672.402} C_VEL
LIN {X 0,Y 502.938,Z 357.836,A -85,B 0,C 180,E1 -5675.613,E2 -5675.613} C_VEL
LIN {X 0,Y 502.906,Z 357.844,A -85,B 0,C 180,E1 -5678.033,E2 -5678.033} C_VEL
LIN {X 0,Y 502.882,Z 357.846,A -85,B 0,C 180,E1 -5681.283,E2 -5681.283} C_VEL
LIN {X 0,Y 502.849,Z 357.85,A -85,B 0,C 180,E1 -5684.571,E2 -5684.571} C_VEL
LIN {X 0,Y 502.866,Z 357.849,A -85,B 0,C 180,E1 -5687.907,E2 -5687.907} C_VEL
LIN {X 0,Y 502.833,Z 357.847,A -85,B 0,C 180,E1 -5690.536,E2 -5690.536} C_VEL
LIN {X 0,Y 502.795,Z 357.857,A -85,B 0,C 180,E1 -5693.04,E2 -5693.04} C_VEL
LIN {X 0,Y 502.844,Z 357.848,A -85,B 0,C 180,E1 -5695.675,E2 -5695.675} C_VEL
LIN {X 0,Y 502.844,Z 357.849,A -85,B 0,C 180,E1 -5698.372,E2 -5698.372} C_VEL
LIN {X 0,Y 502.797,Z 357.857,A -85,B 0,C 180,E1 -5701.499,E2 -5701.499} C_VEL
LIN {X 0,Y 502.807,Z 357.852,A -85,B 0,C 180,E1 -5703.994,E2 -5703.994} C_VEL
LIN {X 0,Y 502.781,Z 357.855,A -85,B 0,C 180,E1 -5707.178,E2 -5707.178} C_VEL
LIN {X 0,Y 502.791,Z 357.855,A -85,B 0,C 180,E1 -5710.015,E2 -5710.015} C_VEL
LIN {X 0,Y 502.806,Z 357.851,A -85,B 0,C 180,E1 -5712.199,E2 -5712.199} C_VEL
LIN {X 0,Y 502.803,Z 357.853,A -85,B 0,C 180,E1 -5715.468,E2 -5715.468} C_VEL
LIN {X 0,Y 502.822,Z 357.85,A -85,B 0,C 180,E1 -5718.934,E2 -5718.934} C_VEL
LIN {X 0,Y 502.796,Z 357.852,A -85,B 0,C 180,E1 -5722.046,E2 -5722.046} C_VEL
LIN {X 0,Y 502.802,Z 357.855,A -85,B 0,C 180,E1 -5725.034,E2 -5725.034} C_VEL
LIN {X 0,Y 502.786,Z 357.858,A -85,B 0,C 180,E1 -5727.915,E2 -5727.915} C_VEL
LIN {X 0,Y 502.827,Z 357.85,A -85,B 0,C 180,E1 -5730.712,E2 -5730.712} C_VEL
LIN {X 0,Y 502.865,Z 357.845,A -85,B 0,C 180,E1 -5733.439,E2 -5733.439} C_VEL
LIN {X 0,Y 502.795,Z 357.855,A -85,B 0,C 180,E1 -5736.086,E2 -5736.086} C_VEL
LIN {X 0,Y 502.787,Z 357.855,A -85,B 0,C 180,E1 -5738.689,E2 -5738.689} C_VEL
LIN {X 0,Y 502.833,Z 357.853,A -85,B 0,C 180,E1 -5741.248,E2 -5741.248} C_VEL
LIN {X 0,Y 502.825,Z 357.849,A -85,B 0,C 180,E1 -5743.767,E2 -5743.767} C_VEL
LIN {X 0,Y 502.834,Z 357.851,A -85,B 0,C 180,E1 -5746.255,E2 -5746.255} C_VEL
LIN {X 0,Y 502.896,Z 357.842,A -85,B 0,C 180,E1 -5748.717,E2 -5748.717} C_VEL
LIN {X 0,Y 502.905,Z 357.841,A -85,B 0,C 180,E1 -5751.967,E2 -5751.967} C_VEL
LIN {X 0,Y 502.941,Z 357.837,A -85,B 0,C 180,E1 -5754.386,E2 -5754.386} C_VEL
LIN {X 0,Y 503.027,Z 357.825,A -85,B 0,C 180,E1 -5757.598,E2 -5757.598} C_VEL
LIN {X 0,Y 503.031,Z 357.828,A -85,B 0,C 180,E1 -5760,E2 -5760} C_VEL
LIN {X 0,Y 503.027,Z 357.825,A -85,B 0,C 180,E1 -5762.402,E2 -5762.402} C_VEL
LIN {X 0,Y 502.94,Z 357.834,A -85,B 0,C 180,E1 -5765.613,E2 -5765.613} C_VEL
LIN {X 0,Y 502.903,Z 357.843,A -85,B 0,C 180,E1 -5768.033,E2 -5768.033} C_VEL
LIN {X 0,Y 502.881,Z 357.846,A -85,B 0,C 180,E1 -5771.283,E2 -5771.283} C_VEL
LIN {X 0,Y 502.848,Z 357.85,A -85,B 0,C 180,E1 -5774.571,E2 -5774.571} C_VEL
LIN {X 0,Y 502.825,Z 357.852,A -85,B 0,C 180,E1 -5777.908,E2 -5777.908} C_VEL
LIN {X 0,Y 502.831,Z 357.849,A -85,B 0,C 180,E1 -5780.536,E2 -5780.536} C_VEL
LIN {X 0,Y 502.793,Z 357.857,A -85,B 0,C 180,E1 -5783.041,E2 -5783.041} C_VEL
LIN {X 0,Y 502.842,Z 357.848,A -85,B 0,C 180,E1 -5785.676,E2 -5785.676} C_VEL
LIN {X 0,Y 502.842,Z 357.849,A -85,B 0,C 180,E1 -5788.373,E2 -5788.373} C_VEL
LIN {X 0,Y 502.795,Z 357.857,A -85,B 0,C 180,E1 -5791.499,E2 -5791.499} C_VEL
LIN {X 0,Y 502.807,Z 357.854,A -85,B 0,C 180,E1 -5794.444,E2 -5794.444} C_VEL
LIN {X 0,Y 502.784,Z 357.855,A -85,B 0,C 180,E1 -5797.178,E2 -5797.178} C_VEL
LIN {X 0,Y 502.79,Z 357.857,A -85,B 0,C 180,E1 -5800.015,E2 -5800.015} C_VEL
LIN {X 0,Y 502.805,Z 357.852,A -85,B 0,C 180,E1 -5802.199,E2 -5802.199} C_VEL
LIN {X 0,Y 502.803,Z 357.853,A -85,B 0,C 180,E1 -5805.468,E2 -5805.468} C_VEL
LIN {X 0,Y 502.832,Z 357.851,A -85,B 0,C 180,E1 -5807.864,E2 -5807.864} C_VEL
LIN {X 0,Y 502.803,Z 357.851,A -85,B 0,C 180,E1 -5811.024,E2 -5811.024} C_VEL
LIN {X 0,Y 502.777,Z 357.857,A -85,B 0,C 180,E1 -5814.169,E2 -5814.169} C_VEL
LIN {X 0,Y 502.835,Z 357.846,A -85,B 0,C 180,E1 -5816.993,E2 -5816.993} C_VEL
LIN {X 0,Y 502.797,Z 357.868,A -85,B 0,C 180,E1 -5818.538,E2 -5818.538} C_VEL
LIN {X 0,Y 505.374,Z 369.61,A -85,B 0,C 180,E1 -5821.177,E2 -5821.177} C_VEL
LIN {X 0,Y 505.537,Z 374.775,A -85,B 0,C 180,E1 -5822.243,E2 -5822.243} C_VEL
LIN {X 0,Y 504.712,Z 390.351,A -85,B 0,C 180,E1 -5825.308,E2 -5825.308} C_VEL
LIN {X 0,Y 504.089,Z 404.823,A -85,B 0,C 180,E1 -5828.102,E2 -5828.102} C_VEL
LIN {X 0,Y 503.53,Z 420.565,A -85,B 0,C 180,E1 -5831.064,E2 -5831.064} C_VEL
LIN {X 0,Y 503.133,Z 437.16,A -85,B 0,C 180,E1 -5834.007,E2 -5834.007} C_VEL
LIN {X 0,Y 502.911,Z 447.26,A -85,B 0,C 180,E1 -5835.831,E2 -5835.831} C_VEL
LIN {X 0,Y 504.365,Z 460.503,A -85,B 0,C 180,E1 -5836.143,E2 -5836.143} C_VEL
LIN {X 0,Y 504.14,Z 474.003,A -85,B 0,C 180,E1 -5836.599,E2 -5836.599} C_VEL
LIN {X 0,Y 503.868,Z 486.5,A -85,B 0,C 180,E1 -5837.2,E2 -5837.2} C_VEL
LIN {X 0,Y 503.594,Z 497.876,A -85,B 0,C 180,E1 -5837.917,E2 -5837.917} C_VEL
LIN {X 0,Y 503.218,Z 508.157,A -85,B 0,C 180,E1 -5838.725,E2 -5838.725} C_VEL
LIN {X 0,Y 502.891,Z 518.525,A -85,B 0,C 180,E1 -5839.736,E2 -5839.736} C_VEL
LIN {X 0,Y 502.644,Z 526.947,A -85,B 0,C 180,E1 -5840.747,E2 -5840.747} C_VEL
LIN {X 0,Y 502.438,Z 535.18,A -85,B 0,C 180,E1 -5841.959,E2 -5841.959} C_VEL
LIN {X 0,Y 502.316,Z 541.996,A -85,B 0,C 180,E1 -5843.21,E2 -5843.21} C_VEL
LIN {X 0,Y 502.282,Z 547.047,A -85,B 0,C 180,E1 -5844.379,E2 -5844.379} C_VEL
LIN {X 0,Y 502.178,Z 551.101,A -85,B 0,C 180,E1 -5845.585,E2 -5845.585} C_VEL
LIN {X 0,Y 502.182,Z 554.094,A -85,B 0,C 180,E1 -5846.791,E2 -5846.791} C_VEL
LIN {X 0,Y 502.122,Z 555.52,A -85,B 0,C 180,E1 -5847.594,E2 -5847.594} C_VEL
LIN {X 0,Y 502.02,Z 557.138,A -85,B 0,C 180,E1 -5849.198,E2 -5849.198} C_VEL
LIN {X 0,Y 502.017,Z 557.351,A -85,B 0,C 180,E1 -5850,E2 -5850} C_VEL
LIN {X 0,Y 502.021,Z 557.124,A -85,B 0,C 180,E1 -5850.802,E2 -5850.802} C_VEL
LIN {X 0,Y 502.122,Z 555.478,A -85,B 0,C 180,E1 -5852.407,E2 -5852.407} C_VEL
LIN {X 0,Y 502.182,Z 554.038,A -85,B 0,C 180,E1 -5853.209,E2 -5853.209} C_VEL
LIN {X 0,Y 502.178,Z 551.013,A -85,B 0,C 180,E1 -5854.415,E2 -5854.415} C_VEL
LIN {X 0,Y 502.281,Z 546.925,A -85,B 0,C 180,E1 -5855.621,E2 -5855.621} C_VEL
LIN {X 0,Y 502.332,Z 540.713,A -85,B 0,C 180,E1 -5857.012,E2 -5857.012} C_VEL
LIN {X 0,Y 502.495,Z 533.721,A -85,B 0,C 180,E1 -5858.242,E2 -5858.242} C_VEL
LIN {X 0,Y 502.708,Z 525.138,A -85,B 0,C 180,E1 -5859.455,E2 -5859.455} C_VEL
LIN {X 0,Y 502.954,Z 516.276,A -85,B 0,C 180,E1 -5860.466,E2 -5860.466} C_VEL
LIN {X 0,Y 503.321,Z 505.359,A -85,B 0,C 180,E1 -5861.477,E2 -5861.477} C_VEL
LIN {X 0,Y 503.575,Z 494.789,A -85,B 0,C 180,E1 -5862.264,E2 -5862.264} C_VEL
LIN {X 0,Y 503.851,Z 483.106,A -85,B 0,C 180,E1 -5862.947,E2 -5862.947} C_VEL
LIN {X 0,Y 504.174,Z 470.53,A -85,B 0,C 180,E1 -5863.503,E2 -5863.503} C_VEL
LIN {X 0,Y 504.269,Z 458.404,A -85,B 0,C 180,E1 -5863.885,E2 -5863.885} C_VEL
LIN {X 0,Y 502.847,Z 446.579,A -85,B 0,C 180,E1 -5864.158,E2 -5864.158} C_VEL
LIN {X 0,Y 503.247,Z 429.135,A -85,B 0,C 180,E1 -5867.263,E2 -5867.263} C_VEL
LIN {X 0,Y 503.721,Z 411.947,A -85,B 0,C 180,E1 -5870.414,E2 -5870.414} C_VEL
LIN {X 0,Y 504.327,Z 396.425,A -85,B 0,C 180,E1 -5873.404,E2 -5873.404} C_VEL
LIN {X 0,Y 505.22,Z 381.6,A -85,B 0,C 180,E1 -5876.433,E2 -5876.433} C_VEL
LIN {X 0,Y 505.827,Z 372.074,A -85,B 0,C 180,E1 -5878.526,E2 -5878.526} C_VEL
LIN {X 0,Y 504.275,Z 364.171,A -85,B 0,C 180,E1 -5880.594,E2 -5880.594} C_VEL
LIN {X 0,Y 502.828,Z 357.854,A -85,B 0,C 180,E1 -5882.496,E2 -5882.496} C_VEL
LIN {X 0,Y 502.802,Z 357.858,A -85,B 0,C 180,E1 -5884.966,E2 -5884.966} C_VEL
LIN {X 0,Y 502.795,Z 357.858,A -85,B 0,C 180,E1 -5887.954,E2 -5887.954} C_VEL
LIN {X 0,Y 502.823,Z 357.854,A -85,B 0,C 180,E1 -5891.066,E2 -5891.066} C_VEL
LIN {X 0,Y 502.785,Z 357.859,A -85,B 0,C 180,E1 -5893.376,E2 -5893.376} C_VEL
LIN {X 0,Y 502.793,Z 357.858,A -85,B 0,C 180,E1 -5895.661,E2 -5895.661} C_VEL
LIN {X 0,Y 502.827,Z 357.854,A -85,B 0,C 180,E1 -5898.935,E2 -5898.935} C_VEL
LIN {X 0,Y 502.8,Z 357.857,A -85,B 0,C 180,E1 -5902.047,E2 -5902.047} C_VEL
LIN {X 0,Y 502.81,Z 357.856,A -85,B 0,C 180,E1 -5905.035,E2 -5905.035} C_VEL
LIN {X 0,Y 502.789,Z 357.86,A -85,B 0,C 180,E1 -5907.916,E2 -5907.916} C_VEL
LIN {X 0,Y 502.819,Z 357.964,A -85,B 0,C 180,E1 -5908.576,E2 -5908.576} C_VEL
LIN {X 0,Y 503.208,Z 360.685,A -85,B 0,C 180,E1 -5909.988,E2 -5909.988} C_VEL
LIN {X 0,Y 503.094,Z 365.866,A -85,B 0,C 180,E1 -5912.549,E2 -5912.549} C_VEL
LIN {X 0,Y 502.927,Z 371.469,A -85,B 0,C 180,E1 -5915.275,E2 -5915.275} C_VEL
LIN {X 0,Y 502.804,Z 376.76,A -85,B 0,C 180,E1 -5917.828,E2 -5917.828} C_VEL
LIN {X 0,Y 502.677,Z 382.119,A -85,B 0,C 180,E1 -5920.394,E2 -5920.394} C_VEL
LIN {X 0,Y 502.583,Z 387.456,A -85,B 0,C 180,E1 -5922.923,E2 -5922.923} C_VEL
LIN {X 0,Y 502.475,Z 392.816,A -85,B 0,C 180,E1 -5925.418,E2 -5925.418} C_VEL
LIN {X 0,Y 502.39,Z 399.934,A -85,B 0,C 180,E1 -5928.706,E2 -5928.706} C_VEL
LIN {X 0,Y 502.31,Z 406.075,A -85,B 0,C 180,E1 -5931.502,E2 -5931.502} C_VEL
LIN {X 0,Y 503.272,Z 413.15,A -85,B 0,C 180,E1 -5931.821,E2 -5931.821} C_VEL
LIN {X 0,Y 503.177,Z 422.061,A -85,B 0,C 180,E1 -5932.304,E2 -5932.304} C_VEL
LIN {X 0,Y 503.018,Z 430.563,A -85,B 0,C 180,E1 -5932.924,E2 -5932.924} C_VEL
LIN {X 0,Y 502.824,Z 437.552,A -85,B 0,C 180,E1 -5933.58,E2 -5933.58} C_VEL
LIN {X 0,Y 502.608,Z 444.287,A -85,B 0,C 180,E1 -5934.383,E2 -5934.383} C_VEL
LIN {X 0,Y 502.517,Z 449.566,A -85,B 0,C 180,E1 -5935.186,E2 -5935.186} C_VEL
LIN {X 0,Y 502.436,Z 453.722,A -85,B 0,C 180,E1 -5935.99,E2 -5935.99} C_VEL
LIN {X 0,Y 502.341,Z 456.946,A -85,B 0,C 180,E1 -5936.792,E2 -5936.792} C_VEL
LIN {X 0,Y 502.216,Z 459.369,A -85,B 0,C 180,E1 -5937.594,E2 -5937.594} C_VEL
LIN {X 0,Y 502.141,Z 461.051,A -85,B 0,C 180,E1 -5938.396,E2 -5938.396} C_VEL
LIN {X 0,Y 502.115,Z 462.039,A -85,B 0,C 180,E1 -5939.198,E2 -5939.198} C_VEL
LIN {X 0,Y 502.106,Z 462.361,A -85,B 0,C 180,E1 -5940,E2 -5940} C_VEL
LIN {X 0,Y 502.105,Z 462.025,A -85,B 0,C 180,E1 -5940.802,E2 -5940.802} C_VEL
LIN {X 0,Y 502.123,Z 461.024,A -85,B 0,C 180,E1 -5941.604,E2 -5941.604} C_VEL
LIN {X 0,Y 502.336,Z 458.197,A -85,B 0,C 180,E1 -5942.807,E2 -5942.807} C_VEL
LIN {X 0,Y 502.462,Z 455.38,A -85,B 0,C 180,E1 -5943.609,E2 -5943.609} C_VEL
LIN {X 0,Y 502.49,Z 450.63,A -85,B 0,C 180,E1 -5944.613,E2 -5944.613} C_VEL
LIN {X 0,Y 502.589,Z 444.219,A -85,B 0,C 180,E1 -5945.617,E2 -5945.617} C_VEL
LIN {X 0,Y 502.669,Z 437.5,A -85,B 0,C 180,E1 -5946.422,E2 -5946.422} C_VEL
LIN {X 0,Y 502.875,Z 429.904,A -85,B 0,C 180,E1 -5947.127,E2 -5947.127} C_VEL
LIN {X 0,Y 503.044,Z 421.522,A -85,B 0,C 180,E1 -5947.728,E2 -5947.728} C_VEL
LIN {X 0,Y 503.075,Z 411.957,A -85,B 0,C 180,E1 -5948.233,E2 -5948.233} C_VEL
LIN {X 0,Y 502.216,Z 405.045,A -85,B 0,C 180,E1 -5948.526,E2 -5948.526} C_VEL
LIN {X 0,Y 502.243,Z 397.995,A -85,B 0,C 180,E1 -5951.613,E2 -5951.613} C_VEL
LIN {X 0,Y 502.334,Z 390.155,A -85,B 0,C 180,E1 -5955.124,E2 -5955.124} C_VEL
LIN {X 0,Y 502.455,Z 384.069,A -85,B 0,C 180,E1 -5957.984,E2 -5957.984} C_VEL
LIN {X 0,Y 502.502,Z 378.671,A -85,B 0,C 180,E1 -5960.466,E2 -5960.466} C_VEL
LIN {X 0,Y 502.589,Z 373.093,A -85,B 0,C 180,E1 -5963.051,E2 -5963.051} C_VEL
LIN {X 0,Y 502.73,Z 367.462,A -85,B 0,C 180,E1 -5965.682,E2 -5965.682} C_VEL
LIN {X 0,Y 502.828,Z 361.774,A -85,B 0,C 180,E1 -5968.374,E2 -5968.374} C_VEL
LIN {X 0,Y 502.947,Z 357.838,A -85,B 0,C 180,E1 -5970.318,E2 -5970.318} C_VEL
LIN {X 0,Y 502.811,Z 357.851,A -85,B 0,C 180,E1 -5973.994,E2 -5973.994} C_VEL
LIN {X 0,Y 502.785,Z 357.855,A -85,B 0,C 180,E1 -5977.178,E2 -5977.178} C_VEL
LIN {X 0,Y 502.792,Z 357.855,A -85,B 0,C 180,E1 -5980.015,E2 -5980.015} C_VEL
LIN {X 0,Y 502.806,Z 357.851,A -85,B 0,C 180,E1 -5982.199,E2 -5982.199} C_VEL
LIN {X 0,Y 502.805,Z 357.852,A -85,B 0,C 180,E1 -5985.468,E2 -5985.468} C_VEL
LIN {X 0,Y 502.834,Z 357.852,A -85,B 0,C 180,E1 -5987.864,E2 -5987.864} C_VEL
LIN {X 0,Y 502.805,Z 357.856,A -85,B 0,C 180,E1 -5991.024,E2 -5991.024} C_VEL
LIN {X 0,Y 502.778,Z 357.856,A -85,B 0,C 180,E1 -5994.169,E2 -5994.169} C_VEL
LIN {X 0,Y 502.802,Z 357.851,A -85,B 0,C 180,E1 -5996.406,E2 -5996.406} C_VEL
LIN {X 0,Y 502.151,Z 357.934,A -85,B 0,C 180,E1 -5997.074,E2 -5997.074} C_VEL
LIN {X 0,Y 499.305,Z 358.293,A -85,B 0,C 180,E1 -5998.159,E2 -5998.159} C_VEL
LIN {X 0,Y 496.889,Z 358.596,A -85,B 0,C 180,E1 -5999.033,E2 -5999.033} C_VEL
LIN {X 0,Y 495.852,Z 358.723,A -85,B 0,C 180,E1 -5999.708,E2 -5999.708} C_VEL
LIN {X 0,Y 495.767,Z 358.732,A -85,B 0,C 180,E1 -5999.937,E2 -5999.937} C_VEL
LIN {X 0,Y 495.818,Z 358.725,A -85,B 0,C 180,E1 -6003.026,E2 -6003.026} C_VEL
LIN {X 0,Y 495.737,Z 358.732,A -85,B 0,C 180,E1 -6005.724,E2 -6005.724} C_VEL
LIN {X 0,Y 495.747,Z 358.733,A -85,B 0,C 180,E1 -6008.371,E2 -6008.371} C_VEL
LIN {X 0,Y 495.788,Z 358.729,A -85,B 0,C 180,E1 -6010.972,E2 -6010.972} C_VEL
LIN {X 0,Y 495.782,Z 358.728,A -85,B 0,C 180,E1 -6013.53,E2 -6013.53} C_VEL
LIN {X 0,Y 495.798,Z 358.727,A -85,B 0,C 180,E1 -6016.056,E2 -6016.056} C_VEL
LIN {X 0,Y 495.856,Z 358.718,A -85,B 0,C 180,E1 -6018.555,E2 -6018.555} C_VEL
LIN {X 0,Y 495.877,Z 358.717,A -85,B 0,C 180,E1 -6021.852,E2 -6021.852} C_VEL
LIN {X 0,Y 495.894,Z 358.715,A -85,B 0,C 180,E1 -6024.306,E2 -6024.306} C_VEL
LIN {X 0,Y 495.997,Z 358.7,A -85,B 0,C 180,E1 -6027.564,E2 -6027.564} C_VEL
LIN {X 0,Y 496.009,Z 358.699,A -85,B 0,C 180,E1 -6030.812,E2 -6030.812} C_VEL
LIN {X 0,Y 495.845,Z 358.723,A -85,B 0,C 180,E1 -6033.25,E2 -6033.25} C_VEL
LIN {X 0,Y 495.865,Z 358.719,A -85,B 0,C 180,E1 -6036.51,E2 -6036.51} C_VEL
LIN {X 0,Y 495.846,Z 358.717,A -85,B 0,C 180,E1 -6038.97,E2 -6038.97} C_VEL
LIN {X 0,Y 495.832,Z 358.721,A -85,B 0,C 180,E1 -6042.035,E2 -6042.035} C_VEL
LIN {X 0,Y 495.828,Z 358.722,A -85,B 0,C 180,E1 -6045.452,E2 -6045.452} C_VEL
LIN {X 0,Y 495.811,Z 358.725,A -85,B 0,C 180,E1 -6048.247,E2 -6048.247} C_VEL
LIN {X 0,Y 495.778,Z 358.727,A -85,B 0,C 180,E1 -6050.756,E2 -6050.756} C_VEL
LIN {X 0,Y 495.752,Z 358.733,A -85,B 0,C 180,E1 -6053.387,E2 -6053.387} C_VEL
LIN {X 0,Y 495.795,Z 358.729,A -85,B 0,C 180,E1 -6056.068,E2 -6056.068} C_VEL
LIN {X 0,Y 495.776,Z 358.727,A -85,B 0,C 180,E1 -6058.815,E2 -6058.815} C_VEL
LIN {X 0,Y 495.76,Z 358.731,A -85,B 0,C 180,E1 -6061.725,E2 -6061.725} C_VEL
LIN {X 0,Y 495.772,Z 358.731,A -85,B 0,C 180,E1 -6064.694,E2 -6064.694} C_VEL
LIN {X 0,Y 495.733,Z 358.735,A -85,B 0,C 180,E1 -6067.561,E2 -6067.561} C_VEL
LIN {X 0,Y 495.769,Z 358.728,A -85,B 0,C 180,E1 -6070.7,E2 -6070.7} C_VEL
LIN {X 0,Y 495.737,Z 358.732,A -85,B 0,C 180,E1 -6074.001,E2 -6074.001} C_VEL
LIN {X 0,Y 495.728,Z 358.734,A -85,B 0,C 180,E1 -6077.117,E2 -6077.117} C_VEL
LIN {X 0,Y 495.761,Z 358.732,A -85,B 0,C 180,E1 -6079.953,E2 -6079.953} C_VEL
LIN {X 0,Y 495.73,Z 358.733,A -85,B 0,C 180,E1 -6082.553,E2 -6082.553} C_VEL
LIN {X 0,Y 495.781,Z 358.727,A -85,B 0,C 180,E1 -6085.457,E2 -6085.457} C_VEL
LIN {X 0,Y 495.758,Z 358.733,A -85,B 0,C 180,E1 -6088.364,E2 -6088.364} C_VEL
LIN {X 0,Y 495.79,Z 358.729,A -85,B 0,C 180,E1 -6091.507,E2 -6091.507} C_VEL
LIN {X 0,Y 495.794,Z 358.724,A -85,B 0,C 180,E1 -6093.932,E2 -6093.932} C_VEL
LIN {X 0,Y 495.769,Z 358.729,A -85,B 0,C 180,E1 -6097.137,E2 -6097.137} C_VEL
LIN {X 0,Y 495.781,Z 358.73,A -85,B 0,C 180,E1 -6100.11,E2 -6100.11} C_VEL
LIN {X 0,Y 495.79,Z 358.728,A -85,B 0,C 180,E1 -6102.681,E2 -6102.681} C_VEL
LIN {X 0,Y 495.793,Z 358.726,A -85,B 0,C 180,E1 -6105.217,E2 -6105.217} C_VEL
LIN {X 0,Y 495.871,Z 358.718,A -85,B 0,C 180,E1 -6108.555,E2 -6108.555} C_VEL
LIN {X 0,Y 495.877,Z 358.717,A -85,B 0,C 180,E1 -6111.852,E2 -6111.852} C_VEL
LIN {X 0,Y 495.898,Z 358.713,A -85,B 0,C 180,E1 -6114.306,E2 -6114.306} C_VEL
LIN {X 0,Y 495.996,Z 358.7,A -85,B 0,C 180,E1 -6117.564,E2 -6117.564} C_VEL
LIN {X 0,Y 496.002,Z 358.704,A -85,B 0,C 180,E1 -6120,E2 -6120} C_VEL
LIN {X 0,Y 495.996,Z 358.701,A -85,B 0,C 180,E1 -6122.436,E2 -6122.436} C_VEL
LIN {X 0,Y 495.898,Z 358.712,A -85,B 0,C 180,E1 -6125.693,E2 -6125.693} C_VEL
LIN {X 0,Y 495.875,Z 358.72,A -85,B 0,C 180,E1 -6128.148,E2 -6128.148} C_VEL
LIN {X 0,Y 495.855,Z 358.721,A -85,B 0,C 180,E1 -6131.445,E2 -6131.445} C_VEL
LIN {X 0,Y 495.793,Z 358.729,A -85,B 0,C 180,E1 -6134.783,E2 -6134.783} C_VEL
LIN {X 0,Y 495.768,Z 358.727,A -85,B 0,C 180,E1 -6137.319,E2 -6137.319} C_VEL
LIN {X 0,Y 495.78,Z 358.732,A -85,B 0,C 180,E1 -6139.89,E2 -6139.89} C_VEL
LIN {X 0,Y 495.762,Z 358.733,A -85,B 0,C 180,E1 -6142.861,E2 -6142.861} C_VEL
LIN {X 0,Y 495.793,Z 358.727,A -85,B 0,C 180,E1 -6146.068,E2 -6146.068} C_VEL
LIN {X 0,Y 495.774,Z 358.727,A -85,B 0,C 180,E1 -6148.815,E2 -6148.815} C_VEL
LIN {X 0,Y 495.758,Z 358.734,A -85,B 0,C 180,E1 -6151.725,E2 -6151.725} C_VEL
LIN {X 0,Y 495.777,Z 358.731,A -85,B 0,C 180,E1 -6154.695,E2 -6154.695} C_VEL
LIN {X 0,Y 495.734,Z 358.733,A -85,B 0,C 180,E1 -6157.561,E2 -6157.561} C_VEL
LIN {X 0,Y 495.768,Z 358.728,A -85,B 0,C 180,E1 -6160.7,E2 -6160.7} C_VEL
LIN {X 0,Y 495.737,Z 358.734,A -85,B 0,C 180,E1 -6163.695,E2 -6163.695} C_VEL
LIN {X 0,Y 495.737,Z 358.737,A -85,B 0,C 180,E1 -6166.305,E2 -6166.305} C_VEL
LIN {X 0,Y 495.769,Z 358.729,A -85,B 0,C 180,E1 -6169.3,E2 -6169.3} C_VEL
LIN {X 0,Y 495.731,Z 358.732,A -85,B 0,C 180,E1 -6172.438,E2 -6172.438} C_VEL
LIN {X 0,Y 495.78,Z 358.727,A -85,B 0,C 180,E1 -6175.457,E2 -6175.457} C_VEL
LIN {X 0,Y 495.766,Z 358.906,A -85,B 0,C 180,E1 -6178.273,E2 -6178.273} C_VEL
LIN {X 0,Y 498.165,Z 369.685,A -85,B 0,C 180,E1 -6180.747,E2 -6180.747} C_VEL
LIN {X 0,Y 498.747,Z 374.726,A -85,B 0,C 180,E1 -6181.832,E2 -6181.832} C_VEL
LIN {X 0,Y 497.783,Z 391.306,A -85,B 0,C 180,E1 -6185.164,E2 -6185.164} C_VEL
LIN {X 0,Y 497.126,Z 405.76,A -85,B 0,C 180,E1 -6187.998,E2 -6187.998} C_VEL
LIN {X 0,Y 496.509,Z 421.406,A -85,B 0,C 180,E1 -6191,E2 -6191} C_VEL
LIN {X 0,Y 496.107,Z 436.527,A -85,B 0,C 180,E1 -6193.753,E2 -6193.753} C_VEL
LIN {X 0,Y 495.878,Z 446.975,A -85,B 0,C 180,E1 -6195.666,E2 -6195.666} C_VEL
LIN {X 0,Y 497.364,Z 459.694,A -85,B 0,C 180,E1 -6195.97,E2 -6195.97} C_VEL
LIN {X 0,Y 497.184,Z 472.652,A -85,B 0,C 180,E1 -6196.408,E2 -6196.408} C_VEL
LIN {X 0,Y 496.891,Z 483.64,A -85,B 0,C 180,E1 -6196.92,E2 -6196.92} C_VEL
LIN {X 0,Y 496.629,Z 495.142,A -85,B 0,C 180,E1 -6197.618,E2 -6197.618} C_VEL
LIN {X 0,Y 496.287,Z 506.092,A -85,B 0,C 180,E1 -6198.462,E2 -6198.462} C_VEL
LIN {X 0,Y 495.93,Z 515.792,A -85,B 0,C 180,E1 -6199.384,E2 -6199.384} C_VEL
LIN {X 0,Y 495.627,Z 524.628,A -85,B 0,C 180,E1 -6200.409,E2 -6200.409} C_VEL
LIN {X 0,Y 495.432,Z 533.204,A -85,B 0,C 180,E1 -6201.639,E2 -6201.639} C_VEL
LIN {X 0,Y 495.248,Z 540.17,A -85,B 0,C 180,E1 -6202.888,E2 -6202.888} C_VEL
LIN {X 0,Y 495.191,Z 546.362,A -85,B 0,C 180,E1 -6204.298,E2 -6204.298} C_VEL
LIN {X 0,Y 495.076,Z 550.429,A -85,B 0,C 180,E1 -6205.522,E2 -6205.522} C_VEL
LIN {X 0,Y 495.116,Z 553.433,A -85,B 0,C 180,E1 -6206.745,E2 -6206.745} C_VEL
LIN {X 0,Y 495.058,Z 554.864,A -85,B 0,C 180,E1 -6207.559,E2 -6207.559} C_VEL
LIN {X 0,Y 494.95,Z 556.48,A -85,B 0,C 180,E1 -6209.186,E2 -6209.186} C_VEL
LIN {X 0,Y 494.948,Z 556.692,A -85,B 0,C 180,E1 -6210,E2 -6210} C_VEL
LIN {X 0,Y 494.951,Z 556.461,A -85,B 0,C 180,E1 -6210.814,E2 -6210.814} C_VEL
LIN {X 0,Y 494.982,Z 555.832,A -85,B 0,C 180,E1 -6211.627,E2 -6211.627} C_VEL
LIN {X 0,Y 495.058,Z 554.802,A -85,B 0,C 180,E1 -6212.441,E2 -6212.441} C_VEL
LIN {X 0,Y 495.133,Z 553.353,A -85,B 0,C 180,E1 -6213.255,E2 -6213.255} C_VEL
LIN {X 0,Y 495.095,Z 550.308,A -85,B 0,C 180,E1 -6214.478,E2 -6214.478} C_VEL
LIN {X 0,Y 495.208,Z 545.028,A -85,B 0,C 180,E1 -6215.992,E2 -6215.992} C_VEL
LIN {X 0,Y 495.274,Z 538.807,A -85,B 0,C 180,E1 -6217.337,E2 -6217.337} C_VEL
LIN {X 0,Y 495.454,Z 531.618,A -85,B 0,C 180,E1 -6218.566,E2 -6218.566} C_VEL
LIN {X 0,Y 495.658,Z 522.602,A -85,B 0,C 180,E1 -6219.797,E2 -6219.797} C_VEL
LIN {X 0,Y 495.977,Z 513.352,A -85,B 0,C 180,E1 -6220.822,E2 -6220.822} C_VEL
LIN {X 0,Y 496.317,Z 503.089,A -85,B 0,C 180,E1 -6221.745,E2 -6221.745} C_VEL
LIN {X 0,Y 496.636,Z 491.978,A -85,B 0,C 180,E1 -6222.546,E2 -6222.546} C_VEL
LIN {X 0,Y 496.962,Z 479.782,A -85,B 0,C 180,E1 -6223.234,E2 -6223.234} C_VEL
LIN {X 0,Y 497.258,Z 466.73,A -85,B 0,C 180,E1 -6223.772,E2 -6223.772} C_VEL
LIN {X 0,Y 497.174,Z 458.237,A -85,B 0,C 180,E1 -6224.035,E2 -6224.035} C_VEL
LIN {X 0,Y 495.805,Z 446.268,A -85,B 0,C 180,E1 -6224.311,E2 -6224.311} C_VEL
LIN {X 0,Y 496.184,Z 429.816,A -85,B 0,C 180,E1 -6227.304,E2 -6227.304} C_VEL
LIN {X 0,Y 496.675,Z 413.906,A -85,B 0,C 180,E1 -6230.284,E2 -6230.284} C_VEL
LIN {X 0,Y 497.293,Z 399.171,A -85,B 0,C 180,E1 -6233.163,E2 -6233.163} C_VEL
LIN {X 0,Y 498.186,Z 384.808,A -85,B 0,C 180,E1 -6236.158,E2 -6236.158} C_VEL
LIN {X 0,Y 498.971,Z 375.789,A -85,B 0,C 180,E1 -6238.154,E2 -6238.154} C_VEL
LIN {X 0,Y 498.705,Z 371.921,A -85,B 0,C 180,E1 -6239.104,E2 -6239.104} C_VEL
LIN {X 0,Y 497.174,Z 364.864,A -85,B 0,C 180,E1 -6241.062,E2 -6241.062} C_VEL
LIN {X 0,Y 495.797,Z 358.728,A -85,B 0,C 180,E1 -6243.026,E2 -6243.026} C_VEL
LIN {X 0,Y 495.722,Z 358.74,A -85,B 0,C 180,E1 -6246.089,E2 -6246.089} C_VEL
LIN {X 0,Y 495.765,Z 358.733,A -85,B 0,C 180,E1 -6248.768,E2 -6248.768} C_VEL
LIN {X 0,Y 495.78,Z 358.731,A -85,B 0,C 180,E1 -6251.779,E2 -6251.779} C_VEL
LIN {X 0,Y 495.752,Z 358.735,A -85,B 0,C 180,E1 -6255.139,E2 -6255.139} C_VEL
LIN {X 0,Y 495.781,Z 358.73,A -85,B 0,C 180,E1 -6258.221,E2 -6258.221} C_VEL
LIN {X 0,Y 495.78,Z 358.732,A -85,B 0,C 180,E1 -6261.23,E2 -6261.23} C_VEL
LIN {X 0,Y 495.758,Z 358.735,A -85,B 0,C 180,E1 -6264.463,E2 -6264.463} C_VEL
LIN {X 0,Y 495.772,Z 358.734,A -85,B 0,C 180,E1 -6267.406,E2 -6267.406} C_VEL
LIN {X 0,Y 495.769,Z 358.923,A -85,B 0,C 180,E1 -6268.273,E2 -6268.273} C_VEL
LIN {X 0,Y 496.231,Z 362.691,A -85,B 0,C 180,E1 -6270.284,E2 -6270.284} C_VEL
LIN {X 0,Y 496.061,Z 368.485,A -85,B 0,C 180,E1 -6273.197,E2 -6273.197} C_VEL
LIN {X 0,Y 495.927,Z 373.611,A -85,B 0,C 180,E1 -6275.734,E2 -6275.734} C_VEL
LIN {X 0,Y 495.779,Z 378.997,A -85,B 0,C 180,E1 -6278.373,E2 -6278.373} C_VEL
LIN {X 0,Y 495.613,Z 386.132,A -85,B 0,C 180,E1 -6281.822,E2 -6281.822} C_VEL
LIN {X 0,Y 495.463,Z 393.301,A -85,B 0,C 180,E1 -6285.207,E2 -6285.207} C_VEL
LIN {X 0,Y 495.349,Z 400.438,A -85,B 0,C 180,E1 -6288.543,E2 -6288.543} C_VEL
LIN {X 0,Y 495.286,Z 406.606,A -85,B 0,C 180,E1 -6291.354,E2 -6291.354} C_VEL
LIN {X 0,Y 496.334,Z 414.357,A -85,B 0,C 180,E1 -6291.706,E2 -6291.706} C_VEL
LIN {X 0,Y 496.209,Z 423.05,A -85,B 0,C 180,E1 -6292.196,E2 -6292.196} C_VEL
LIN {X 0,Y 496.043,Z 431.445,A -85,B 0,C 180,E1 -6292.826,E2 -6292.826} C_VEL
LIN {X 0,Y 495.825,Z 438.334,A -85,B 0,C 180,E1 -6293.489,E2 -6293.489} C_VEL
LIN {X 0,Y 495.601,Z 445.031,A -85,B 0,C 180,E1 -6294.303,E2 -6294.303} C_VEL
LIN {X 0,Y 495.494,Z 450.299,A -85,B 0,C 180,E1 -6295.118,E2 -6295.118} C_VEL
LIN {X 0,Y 495.402,Z 454.435,A -85,B 0,C 180,E1 -6295.933,E2 -6295.933} C_VEL
LIN {X 0,Y 495.293,Z 457.652,A -85,B 0,C 180,E1 -6296.746,E2 -6296.746} C_VEL
LIN {X 0,Y 495.158,Z 460.069,A -85,B 0,C 180,E1 -6297.56,E2 -6297.56} C_VEL
LIN {X 0,Y 495.079,Z 461.744,A -85,B 0,C 180,E1 -6298.373,E2 -6298.373} C_VEL
LIN {X 0,Y 495.05,Z 462.725,A -85,B 0,C 180,E1 -6299.187,E2 -6299.187} C_VEL
LIN {X 0,Y 495.039,Z 463.04,A -85,B 0,C 180,E1 -6300,E2 -6300} C_VEL
LIN {X 0,Y 495.038,Z 462.693,A -85,B 0,C 180,E1 -6300.814,E2 -6300.814} C_VEL
LIN {X 0,Y 495.057,Z 461.68,A -85,B 0,C 180,E1 -6301.627,E2 -6301.627} C_VEL
LIN {X 0,Y 495.294,Z 458.839,A -85,B 0,C 180,E1 -6302.847,E2 -6302.847} C_VEL
LIN {X 0,Y 495.402,Z 456.005,A -85,B 0,C 180,E1 -6303.66,E2 -6303.66} C_VEL
LIN {X 0,Y 495.458,Z 451.24,A -85,B 0,C 180,E1 -6304.678,E2 -6304.678} C_VEL
LIN {X 0,Y 495.57,Z 444.814,A -85,B 0,C 180,E1 -6305.697,E2 -6305.697} C_VEL
LIN {X 0,Y 495.646,Z 438.103,A -85,B 0,C 180,E1 -6306.514,E2 -6306.514} C_VEL
LIN {X 0,Y 495.863,Z 430.965,A -85,B 0,C 180,E1 -6307.192,E2 -6307.192} C_VEL
LIN {X 0,Y 496.056,Z 422.185,A -85,B 0,C 180,E1 -6307.838,E2 -6307.838} C_VEL
LIN {X 0,Y 496.114,Z 412.778,A -85,B 0,C 180,E1 -6308.349,E2 -6308.349} C_VEL
LIN {X 0,Y 495.128,Z 405.338,A -85,B 0,C 180,E1 -6308.674,E2 -6308.674} C_VEL
LIN {X 0,Y 495.176,Z 398.588,A -85,B 0,C 180,E1 -6311.674,E2 -6311.674} C_VEL
LIN {X 0,Y 495.302,Z 390.759,A -85,B 0,C 180,E1 -6315.23,E2 -6315.23} C_VEL
LIN {X 0,Y 495.397,Z 384.374,A -85,B 0,C 180,E1 -6318.186,E2 -6318.186} C_VEL
LIN {X 0,Y 495.462,Z 378.814,A -85,B 0,C 180,E1 -6320.77,E2 -6320.77} C_VEL
LIN {X 0,Y 495.554,Z 373.195,A -85,B 0,C 180,E1 -6323.397,E2 -6323.397} C_VEL
LIN {X 0,Y 495.678,Z 367.561,A -85,B 0,C 180,E1 -6326.074,E2 -6326.074} C_VEL
LIN {X 0,Y 495.813,Z 361.801,A -85,B 0,C 180,E1 -6328.812,E2 -6328.812} C_VEL
LIN {X 0,Y 495.896,Z 358.716,A -85,B 0,C 180,E1 -6330.388,E2 -6330.388} C_VEL
LIN {X 0,Y 495.764,Z 358.728,A -85,B 0,C 180,E1 -6333.564,E2 -6333.564} C_VEL
LIN {X 0,Y 495.737,Z 358.736,A -85,B 0,C 180,E1 -6336.543,E2 -6336.543} C_VEL
LIN {X 0,Y 495.761,Z 358.733,A -85,B 0,C 180,E1 -6339.638,E2 -6339.638} C_VEL
LIN {X 0,Y 495.741,Z 358.733,A -85,B 0,C 180,E1 -6342.507,E2 -6342.507} C_VEL
LIN {X 0,Y 495.753,Z 358.731,A -85,B 0,C 180,E1 -6345.139,E2 -6345.139} C_VEL
LIN {X 0,Y 495.781,Z 358.731,A -85,B 0,C 180,E1 -6348.221,E2 -6348.221} C_VEL
LIN {X 0,Y 495.754,Z 358.733,A -85,B 0,C 180,E1 -6351.408,E2 -6351.408} C_VEL
LIN {X 0,Y 495.752,Z 358.734,A -85,B 0,C 180,E1 -6354.462,E2 -6354.462} C_VEL
LIN {X 0,Y 495.772,Z 358.729,A -85,B 0,C 180,E1 -6357.406,E2 -6357.406} C_VEL
LIN {X 0,Y 495.767,Z 358.732,A -85,B 0,C 180,E1 -6359.937,E2 -6359.937} C_VEL
LIN {X 0,Y 495.109,Z 358.812,A -85,B 0,C 180,E1 -6360.615,E2 -6360.615} C_VEL
LIN {X 0,Y 492.285,Z 359.165,A -85,B 0,C 180,E1 -6361.715,E2 -6361.715} C_VEL
LIN {X 0,Y 489.888,Z 359.464,A -85,B 0,C 180,E1 -6362.602,E2 -6362.602} C_VEL
LIN {X 0,Y 488.848,Z 359.592,A -85,B 0,C 180,E1 -6363.287,E2 -6363.287} C_VEL
LIN {X 0,Y 488.757,Z 359.602,A -85,B 0,C 180,E1 -6363.519,E2 -6363.519} C_VEL
LIN {X 0,Y 488.685,Z 359.615,A -85,B 0,C 180,E1 -6366.254,E2 -6366.254} C_VEL
LIN {X 0,Y 488.75,Z 359.604,A -85,B 0,C 180,E1 -6369.176,E2 -6369.176} C_VEL
LIN {X 0,Y 488.764,Z 359.604,A -85,B 0,C 180,E1 -6371.628,E2 -6371.628} C_VEL
LIN {X 0,Y 488.766,Z 359.602,A -85,B 0,C 180,E1 -6375,E2 -6375} C_VEL
LIN {X 0,Y 488.81,Z 359.597,A -85,B 0,C 180,E1 -6378.388,E2 -6378.388} C_VEL
LIN {X 0,Y 488.821,Z 359.596,A -85,B 0,C 180,E1 -6381.734,E2 -6381.734} C_VEL
LIN {X 0,Y 488.853,Z 359.592,A -85,B 0,C 180,E1 -6384.224,E2 -6384.224} C_VEL
LIN {X 0,Y 488.965,Z 359.576,A -85,B 0,C 180,E1 -6387.529,E2 -6387.529} C_VEL
LIN {X 0,Y 488.959,Z 359.578,A -85,B 0,C 180,E1 -6390.824,E2 -6390.824} C_VEL
LIN {X 0,Y 488.965,Z 359.578,A -85,B 0,C 180,E1 -6392.471,E2 -6392.471} C_VEL
LIN {X 0,Y 488.852,Z 359.591,A -85,B 0,C 180,E1 -6395.776,E2 -6395.776} C_VEL
LIN {X 0,Y 488.821,Z 359.595,A -85,B 0,C 180,E1 -6398.266,E2 -6398.266} C_VEL
LIN {X 0,Y 488.81,Z 359.599,A -85,B 0,C 180,E1 -6401.612,E2 -6401.612} C_VEL
LIN {X 0,Y 488.766,Z 359.604,A -85,B 0,C 180,E1 -6405,E2 -6405} C_VEL
LIN {X 0,Y 488.759,Z 359.602,A -85,B 0,C 180,E1 -6408.442,E2 -6408.442} C_VEL
LIN {X 0,Y 488.711,Z 359.609,A -85,B 0,C 180,E1 -6411.071,E2 -6411.071} C_VEL
LIN {X 0,Y 488.693,Z 359.611,A -85,B 0,C 180,E1 -6413.745,E2 -6413.745} C_VEL
LIN {X 0,Y 488.796,Z 359.598,A -85,B 0,C 180,E1 -6416.944,E2 -6416.944} C_VEL
LIN {X 0,Y 488.713,Z 359.606,A -85,B 0,C 180,E1 -6420.363,E2 -6420.363} C_VEL
LIN {X 0,Y 488.738,Z 359.606,A -85,B 0,C 180,E1 -6423.484,E2 -6423.484} C_VEL
LIN {X 0,Y 488.685,Z 359.614,A -85,B 0,C 180,E1 -6426.354,E2 -6426.354} C_VEL
LIN {X 0,Y 488.705,Z 359.61,A -85,B 0,C 180,E1 -6429.254,E2 -6429.254} C_VEL
LIN {X 0,Y 488.71,Z 359.61,A -85,B 0,C 180,E1 -6431.6,E2 -6431.6} C_VEL
LIN {X 0,Y 488.715,Z 359.611,A -85,B 0,C 180,E1 -6434.801,E2 -6434.801} C_VEL
LIN {X 0,Y 488.694,Z 359.611,A -85,B 0,C 180,E1 -6437.474,E2 -6437.474} C_VEL
LIN {X 0,Y 488.735,Z 359.608,A -85,B 0,C 180,E1 -6439.677,E2 -6439.677} C_VEL
LIN {X 0,Y 488.682,Z 359.613,A -85,B 0,C 180,E1 -6442.841,E2 -6442.841} C_VEL
LIN {X 0,Y 488.733,Z 359.606,A -85,B 0,C 180,E1 -6445.887,E2 -6445.887} C_VEL
LIN {X 0,Y 488.695,Z 359.611,A -85,B 0,C 180,E1 -6448.82,E2 -6448.82} C_VEL
LIN {X 0,Y 488.747,Z 359.605,A -85,B 0,C 180,E1 -6451.671,E2 -6451.671} C_VEL
LIN {X 0,Y 488.75,Z 359.604,A -85,B 0,C 180,E1 -6454.444,E2 -6454.444} C_VEL
LIN {X 0,Y 488.731,Z 359.606,A -85,B 0,C 180,E1 -6457.153,E2 -6457.153} C_VEL
LIN {X 0,Y 488.732,Z 359.608,A -85,B 0,C 180,E1 -6459.811,E2 -6459.811} C_VEL
LIN {X 0,Y 488.737,Z 359.605,A -85,B 0,C 180,E1 -6462.423,E2 -6462.423} C_VEL
LIN {X 0,Y 488.765,Z 359.603,A -85,B 0,C 180,E1 -6465,E2 -6465} C_VEL
LIN {X 0,Y 488.833,Z 359.596,A -85,B 0,C 180,E1 -6468.388,E2 -6468.388} C_VEL
LIN {X 0,Y 488.821,Z 359.597,A -85,B 0,C 180,E1 -6471.734,E2 -6471.734} C_VEL
LIN {X 0,Y 488.858,Z 359.59,A -85,B 0,C 180,E1 -6474.224,E2 -6474.224} C_VEL
LIN {X 0,Y 488.964,Z 359.576,A -85,B 0,C 180,E1 -6477.529,E2 -6477.529} C_VEL
LIN {X 0,Y 488.957,Z 359.578,A -85,B 0,C 180,E1 -6480.824,E2 -6480.824} C_VEL
LIN {X 0,Y 488.964,Z 359.577,A -85,B 0,C 180,E1 -6482.471,E2 -6482.471} C_VEL
LIN {X 0,Y 488.857,Z 359.589,A -85,B 0,C 180,E1 -6485.776,E2 -6485.776} C_VEL
LIN {X 0,Y 488.819,Z 359.598,A -85,B 0,C 180,E1 -6488.266,E2 -6488.266} C_VEL
LIN {X 0,Y 488.809,Z 359.599,A -85,B 0,C 180,E1 -6491.612,E2 -6491.612} C_VEL
LIN {X 0,Y 488.765,Z 359.603,A -85,B 0,C 180,E1 -6495,E2 -6495} C_VEL
LIN {X 0,Y 488.749,Z 359.605,A -85,B 0,C 180,E1 -6498.442,E2 -6498.442} C_VEL
LIN {X 0,Y 488.709,Z 359.61,A -85,B 0,C 180,E1 -6501.071,E2 -6501.071} C_VEL
LIN {X 0,Y 488.691,Z 359.611,A -85,B 0,C 180,E1 -6503.746,E2 -6503.746} C_VEL
LIN {X 0,Y 488.794,Z 359.598,A -85,B 0,C 180,E1 -6506.944,E2 -6506.944} C_VEL
LIN {X 0,Y 488.712,Z 359.608,A -85,B 0,C 180,E1 -6510.363,E2 -6510.363} C_VEL
LIN {X 0,Y 488.738,Z 359.607,A -85,B 0,C 180,E1 -6513.484,E2 -6513.484} C_VEL
LIN {X 0,Y 488.691,Z 359.615,A -85,B 0,C 180,E1 -6516.356,E2 -6516.356} C_VEL
LIN {X 0,Y 488.703,Z 359.608,A -85,B 0,C 180,E1 -6519.254,E2 -6519.254} C_VEL
LIN {X 0,Y 488.725,Z 359.611,A -85,B 0,C 180,E1 -6521.602,E2 -6521.602} C_VEL
LIN {X 0,Y 488.714,Z 359.61,A -85,B 0,C 180,E1 -6524.801,E2 -6524.801} C_VEL
LIN {X 0,Y 488.697,Z 359.61,A -85,B 0,C 180,E1 -6527.475,E2 -6527.475} C_VEL
LIN {X 0,Y 488.735,Z 359.608,A -85,B 0,C 180,E1 -6529.677,E2 -6529.677} C_VEL
LIN {X 0,Y 488.681,Z 359.613,A -85,B 0,C 180,E1 -6532.841,E2 -6532.841} C_VEL
LIN {X 0,Y 488.733,Z 359.605,A -85,B 0,C 180,E1 -6535.887,E2 -6535.887} C_VEL
LIN {X 0,Y 488.738,Z 359.703,A -85,B 0,C 180,E1 -6537.956,E2 -6537.956} C_VEL
LIN {X 0,Y 491.351,Z 371.701,A -85,B 0,C 180,E1 -6540.752,E2 -6540.752} C_VEL
LIN {X 0,Y 491.857,Z 375.707,A -85,B 0,C 180,E1 -6541.634,E2 -6541.634} C_VEL
LIN {X 0,Y 490.961,Z 391.151,A -85,B 0,C 180,E1 -6544.795,E2 -6544.795} C_VEL
LIN {X 0,Y 490.174,Z 406.695,A -85,B 0,C 180,E1 -6547.891,E2 -6547.891} C_VEL
LIN {X 0,Y 489.465,Z 423.28,A -85,B 0,C 180,E1 -6551.125,E2 -6551.125} C_VEL
LIN {X 0,Y 488.998,Z 438.253,A -85,B 0,C 180,E1 -6553.939,E2 -6553.939} C_VEL
LIN {X 0,Y 488.839,Z 446.686,A -85,B 0,C 180,E1 -6555.495,E2 -6555.495} C_VEL
LIN {X 0,Y 490.232,Z 458.851,A -85,B 0,C 180,E1 -6555.788,E2 -6555.788} C_VEL
LIN {X 0,Y 490.302,Z 470.012,A -85,B 0,C 180,E1 -6556.161,E2 -6556.161} C_VEL
LIN {X 0,Y 489.91,Z 482.49,A -85,B 0,C 180,E1 -6556.731,E2 -6556.731} C_VEL
LIN {X 0,Y 489.618,Z 494.232,A -85,B 0,C 180,E1 -6557.443,E2 -6557.443} C_VEL
LIN {X 0,Y 489.212,Z 505.197,A -85,B 0,C 180,E1 -6558.292,E2 -6558.292} C_VEL
LIN {X 0,Y 488.878,Z 514.962,A -85,B 0,C 180,E1 -6559.229,E2 -6559.229} C_VEL
LIN {X 0,Y 488.568,Z 523.845,A -85,B 0,C 180,E1 -6560.269,E2 -6560.269} C_VEL
LIN {X 0,Y 488.361,Z 531.166,A -85,B 0,C 180,E1 -6561.309,E2 -6561.309} C_VEL
LIN {X 0,Y 488.203,Z 538.338,A -85,B 0,C 180,E1 -6562.556,E2 -6562.556} C_VEL
LIN {X 0,Y 488.067,Z 543.836,A -85,B 0,C 180,E1 -6563.75,E2 -6563.75} C_VEL
LIN {X 0,Y 487.973,Z 548.5,A -85,B 0,C 180,E1 -6565.043,E2 -6565.043} C_VEL
LIN {X 0,Y 488.068,Z 550.862,A -85,B 0,C 180,E1 -6565.871,E2 -6565.871} C_VEL
LIN {X 0,Y 488.039,Z 552.77,A -85,B 0,C 180,E1 -6566.698,E2 -6566.698} C_VEL
LIN {X 0,Y 487.995,Z 554.208,A -85,B 0,C 180,E1 -6567.524,E2 -6567.524} C_VEL
LIN {X 0,Y 487.88,Z 555.823,A -85,B 0,C 180,E1 -6569.175,E2 -6569.175} C_VEL
LIN {X 0,Y 487.88,Z 556.033,A -85,B 0,C 180,E1 -6570,E2 -6570} C_VEL
LIN {X 0,Y 487.882,Z 555.799,A -85,B 0,C 180,E1 -6570.825,E2 -6570.825} C_VEL
LIN {X 0,Y 487.996,Z 554.126,A -85,B 0,C 180,E1 -6572.476,E2 -6572.476} C_VEL
LIN {X 0,Y 488.054,Z 552.665,A -85,B 0,C 180,E1 -6573.302,E2 -6573.302} C_VEL
LIN {X 0,Y 487.998,Z 549.6,A -85,B 0,C 180,E1 -6574.543,E2 -6574.543} C_VEL
LIN {X 0,Y 488.131,Z 545.466,A -85,B 0,C 180,E1 -6575.784,E2 -6575.784} C_VEL
LIN {X 0,Y 488.181,Z 539.078,A -85,B 0,C 180,E1 -6577.237,E2 -6577.237} C_VEL
LIN {X 0,Y 488.357,Z 532.111,A -85,B 0,C 180,E1 -6578.483,E2 -6578.483} C_VEL
LIN {X 0,Y 488.521,Z 524.986,A -85,B 0,C 180,E1 -6579.523,E2 -6579.523} C_VEL
LIN {X 0,Y 488.805,Z 516.389,A -85,B 0,C 180,E1 -6580.563,E2 -6580.563} C_VEL
LIN {X 0,Y 489.183,Z 505.731,A -85,B 0,C 180,E1 -6581.603,E2 -6581.603} C_VEL
LIN {X 0,Y 489.506,Z 494.295,A -85,B 0,C 180,E1 -6582.499,E2 -6582.499} C_VEL
LIN {X 0,Y 489.846,Z 482.569,A -85,B 0,C 180,E1 -6583.213,E2 -6583.213} C_VEL
LIN {X 0,Y 490.194,Z 470.02,A -85,B 0,C 180,E1 -6583.79,E2 -6583.79} C_VEL
LIN {X 0,Y 490.219,Z 459.018,A -85,B 0,C 180,E1 -6584.159,E2 -6584.159} C_VEL
LIN {X 0,Y 488.867,Z 447.25,A -85,B 0,C 180,E1 -6584.452,E2 -6584.452} C_VEL
LIN {X 0,Y 488.785,Z 445.701,A -85,B 0,C 180,E1 -6584.521,E2 -6584.521} C_VEL
LIN {X 0,Y 489.24,Z 427.08,A -85,B 0,C 180,E1 -6587.99,E2 -6587.99} C_VEL
LIN {X 0,Y 489.852,Z 410.694,A -85,B 0,C 180,E1 -6591.161,E2 -6591.161} C_VEL
LIN {X 0,Y 490.607,Z 396.283,A -85,B 0,C 180,E1 -6594.096,E2 -6594.096} C_VEL
LIN {X 0,Y 491.708,Z 381.951,A -85,B 0,C 180,E1 -6597.218,E2 -6597.218} C_VEL
LIN {X 0,Y 492.159,Z 376.135,A -85,B 0,C 180,E1 -6598.58,E2 -6598.58} C_VEL
LIN {X 0,Y 491.014,Z 369.406,A -85,B 0,C 180,E1 -6600.401,E2 -6600.401} C_VEL
LIN {X 0,Y 489.031,Z 360.877,A -85,B 0,C 180,E1 -6603.101,E2 -6603.101} C_VEL
LIN {X 0,Y 488.74,Z 359.609,A -85,B 0,C 180,E1 -6603.585,E2 -6603.585} C_VEL
LIN {X 0,Y 488.685,Z 359.616,A -85,B 0,C 180,E1 -6606.355,E2 -6606.355} C_VEL
LIN {X 0,Y 488.703,Z 359.613,A -85,B 0,C 180,E1 -6609.254,E2 -6609.254} C_VEL
LIN {X 0,Y 488.726,Z 359.61,A -85,B 0,C 180,E1 -6611.602,E2 -6611.602} C_VEL
LIN {X 0,Y 488.715,Z 359.612,A -85,B 0,C 180,E1 -6614.801,E2 -6614.801} C_VEL
LIN {X 0,Y 488.698,Z 359.612,A -85,B 0,C 180,E1 -6617.475,E2 -6617.475} C_VEL
LIN {X 0,Y 488.75,Z 359.608,A -85,B 0,C 180,E1 -6620.75,E2 -6620.75} C_VEL
LIN {X 0,Y 488.686,Z 359.615,A -85,B 0,C 180,E1 -6623.869,E2 -6623.869} C_VEL
LIN {X 0,Y 488.742,Z 359.61,A -85,B 0,C 180,E1 -6626.877,E2 -6626.877} C_VEL
LIN {X 0,Y 488.733,Z 359.752,A -85,B 0,C 180,E1 -6627.855,E2 -6627.855} C_VEL
LIN {X 0,Y 489.301,Z 363.271,A -85,B 0,C 180,E1 -6629.82,E2 -6629.82} C_VEL
LIN {X 0,Y 489.112,Z 368.7,A -85,B 0,C 180,E1 -6632.625,E2 -6632.625} C_VEL
LIN {X 0,Y 488.935,Z 374.11,A -85,B 0,C 180,E1 -6635.364,E2 -6635.364} C_VEL
LIN {X 0,Y 488.773,Z 379.487,A -85,B 0,C 180,E1 -6638.047,E2 -6638.047} C_VEL
LIN {X 0,Y 488.625,Z 384.871,A -85,B 0,C 180,E1 -6640.682,E2 -6640.682} C_VEL
LIN {X 0,Y 488.505,Z 390.206,A -85,B 0,C 180,E1 -6643.278,E2 -6643.278} C_VEL
LIN {X 0,Y 488.342,Z 395.588,A -85,B 0,C 180,E1 -6645.838,E2 -6645.838} C_VEL
LIN {X 0,Y 488.31,Z 400.95,A -85,B 0,C 180,E1 -6648.376,E2 -6648.376} C_VEL
LIN {X 0,Y 488.229,Z 406.969,A -85,B 0,C 180,E1 -6651.176,E2 -6651.176} C_VEL
LIN {X 0,Y 489.369,Z 414.623,A -85,B 0,C 180,E1 -6651.535,E2 -6651.535} C_VEL
LIN {X 0,Y 489.228,Z 424.099,A -85,B 0,C 180,E1 -6652.084,E2 -6652.084} C_VEL
LIN {X 0,Y 489.07,Z 432.374,A -85,B 0,C 180,E1 -6652.724,E2 -6652.724} C_VEL
LIN {X 0,Y 488.835,Z 439.186,A -85,B 0,C 180,E1 -6653.395,E2 -6653.395} C_VEL
LIN {X 0,Y 488.597,Z 445.821,A -85,B 0,C 180,E1 -6654.221,E2 -6654.221} C_VEL
LIN {X 0,Y 488.472,Z 451.058,A -85,B 0,C 180,E1 -6655.048,E2 -6655.048} C_VEL
LIN {X 0,Y 488.371,Z 455.168,A -85,B 0,C 180,E1 -6655.874,E2 -6655.874} C_VEL
LIN {X 0,Y 488.247,Z 458.371,A -85,B 0,C 180,E1 -6656.699,E2 -6656.699} C_VEL
LIN {X 0,Y 488.101,Z 460.777,A -85,B 0,C 180,E1 -6657.524,E2 -6657.524} C_VEL
LIN {X 0,Y 488.017,Z 462.443,A -85,B 0,C 180,E1 -6658.35,E2 -6658.35} C_VEL
LIN {X 0,Y 487.985,Z 463.414,A -85,B 0,C 180,E1 -6659.175,E2 -6659.175} C_VEL
LIN {X 0,Y 487.973,Z 463.719,A -85,B 0,C 180,E1 -6660,E2 -6660} C_VEL
LIN {X 0,Y 487.971,Z 463.361,A -85,B 0,C 180,E1 -6660.825,E2 -6660.825} C_VEL
LIN {X 0,Y 487.992,Z 462.337,A -85,B 0,C 180,E1 -6661.651,E2 -6661.651} C_VEL
LIN {X 0,Y 488.253,Z 459.478,A -85,B 0,C 180,E1 -6662.888,E2 -6662.888} C_VEL
LIN {X 0,Y 488.365,Z 454.882,A -85,B 0,C 180,E1 -6664.126,E2 -6664.126} C_VEL
LIN {X 0,Y 488.475,Z 449.489,A -85,B 0,C 180,E1 -6665.159,E2 -6665.159} C_VEL
LIN {X 0,Y 488.561,Z 443.889,A -85,B 0,C 180,E1 -6665.986,E2 -6665.986} C_VEL
LIN {X 0,Y 488.693,Z 437.084,A -85,B 0,C 180,E1 -6666.777,E2 -6666.777} C_VEL
LIN {X 0,Y 488.883,Z 428.644,A -85,B 0,C 180,E1 -6667.538,E2 -6667.538} C_VEL
LIN {X 0,Y 489.148,Z 419.489,A -85,B 0,C 180,E1 -6668.157,E2 -6668.157} C_VEL
LIN {X 0,Y 489.07,Z 412.455,A -85,B 0,C 180,E1 -6668.522,E2 -6668.522} C_VEL
LIN {X 0,Y 488.064,Z 405.631,A -85,B 0,C 180,E1 -6668.827,E2 -6668.827} C_VEL
LIN {X 0,Y 488.126,Z 399.16,A -85,B 0,C 180,E1 -6671.745,E2 -6671.745} C_VEL
LIN {X 0,Y 488.263,Z 391.303,A -85,B 0,C 180,E1 -6675.335,E2 -6675.335} C_VEL
LIN {X 0,Y 488.33,Z 384.548,A -85,B 0,C 180,E1 -6678.459,E2 -6678.459} C_VEL
LIN {X 0,Y 488.419,Z 378.942,A -85,B 0,C 180,E1 -6681.084,E2 -6681.084} C_VEL
LIN {X 0,Y 488.524,Z 373.299,A -85,B 0,C 180,E1 -6683.754,E2 -6683.754} C_VEL
LIN {X 0,Y 488.671,Z 366.682,A -85,B 0,C 180,E1 -6686.915,E2 -6686.915} C_VEL
LIN {X 0,Y 488.914,Z 359.862,A -85,B 0,C 180,E1 -6690.207,E2 -6690.207} C_VEL
LIN {X 0,Y 488.847,Z 359.594,A -85,B 0,C 180,E1 -6690.39,E2 -6690.39} C_VEL
LIN {X 0,Y 488.738,Z 359.605,A -85,B 0,C 180,E1 -6694.113,E2 -6694.113} C_VEL
LIN {X 0,Y 488.686,Z 359.611,A -85,B 0,C 180,E1 -6697.159,E2 -6697.159} C_VEL
LIN {X 0,Y 488.722,Z 359.607,A -85,B 0,C 180,E1 -6700.345,E2 -6700.345} C_VEL
LIN {X 0,Y 488.69,Z 359.609,A -85,B 0,C 180,E1 -6703.654,E2 -6703.654} C_VEL
LIN {X 0,Y 488.696,Z 359.614,A -85,B 0,C 180,E1 -6706.346,E2 -6706.346} C_VEL
LIN {X 0,Y 488.722,Z 359.607,A -85,B 0,C 180,E1 -6708.586,E2 -6708.586} C_VEL
LIN {X 0,Y 488.683,Z 359.612,A -85,B 0,C 180,E1 -6711.8,E2 -6711.8} C_VEL
LIN {X 0,Y 488.727,Z 359.606,A -85,B 0,C 180,E1 -6715.053,E2 -6715.053} C_VEL
LIN {X 0,Y 488.708,Z 359.612,A -85,B 0,C 180,E1 -6718.046,E2 -6718.046} C_VEL
LIN {X 0,Y 488.728,Z 359.607,A -85,B 0,C 180,E1 -6720.73,E2 -6720.73} C_VEL
LIN {X 0,Y 488.757,Z 359.602,A -85,B 0,C 180,E1 -6723.519,E2 -6723.519} C_VEL
LIN {X 0,Y 488.073,Z 359.69,A -85,B 0,C 180,E1 -6724.207,E2 -6724.207} C_VEL
LIN {X 0,Y 485.21,Z 360.044,A -85,B 0,C 180,E1 -6725.324,E2 -6725.324} C_VEL
LIN {X 0,Y 482.791,Z 360.349,A -85,B 0,C 180,E1 -6726.224,E2 -6726.224} C_VEL
LIN {X 0,Y 481.745,Z 360.475,A -85,B 0,C 180,E1 -6726.92,E2 -6726.92} C_VEL
LIN {X 0,Y 481.654,Z 360.486,A -85,B 0,C 180,E1 -6727.155,E2 -6727.155} C_VEL
LIN {X 0,Y 481.7,Z 360.483,A -85,B 0,C 180,E1 -6729.503,E2 -6729.503} C_VEL
LIN {X 0,Y 481.709,Z 360.481,A -85,B 0,C 180,E1 -6732.158,E2 -6732.158} C_VEL
LIN {X 0,Y 481.747,Z 360.478,A -85,B 0,C 180,E1 -6734.776,E2 -6734.776} C_VEL
LIN {X 0,Y 481.755,Z 360.477,A -85,B 0,C 180,E1 -6738.215,E2 -6738.215} C_VEL
LIN {X 0,Y 481.766,Z 360.476,A -85,B 0,C 180,E1 -6741.612,E2 -6741.612} C_VEL
LIN {X 0,Y 481.813,Z 360.469,A -85,B 0,C 180,E1 -6744.139,E2 -6744.139} C_VEL
LIN {X 0,Y 481.932,Z 360.452,A -85,B 0,C 180,E1 -6747.492,E2 -6747.492} C_VEL
LIN {X 0,Y 481.91,Z 360.456,A -85,B 0,C 180,E1 -6750.836,E2 -6750.836} C_VEL
LIN {X 0,Y 481.932,Z 360.454,A -85,B 0,C 180,E1 -6752.507,E2 -6752.507} C_VEL
LIN {X 0,Y 481.813,Z 360.469,A -85,B 0,C 180,E1 -6755.86,E2 -6755.86} C_VEL
LIN {X 0,Y 481.767,Z 360.473,A -85,B 0,C 180,E1 -6758.388,E2 -6758.388} C_VEL
LIN {X 0,Y 481.755,Z 360.476,A -85,B 0,C 180,E1 -6761.785,E2 -6761.785} C_VEL
LIN {X 0,Y 481.747,Z 360.477,A -85,B 0,C 180,E1 -6765.224,E2 -6765.224} C_VEL
LIN {X 0,Y 481.717,Z 360.478,A -85,B 0,C 180,E1 -6768.722,E2 -6768.722} C_VEL
LIN {X 0,Y 481.65,Z 360.492,A -85,B 0,C 180,E1 -6771.395,E2 -6771.395} C_VEL
LIN {X 0,Y 481.678,Z 360.485,A -85,B 0,C 180,E1 -6774.113,E2 -6774.113} C_VEL
LIN {X 0,Y 481.751,Z 360.475,A -85,B 0,C 180,E1 -6777.139,E2 -6777.139} C_VEL
LIN {X 0,Y 481.682,Z 360.487,A -85,B 0,C 180,E1 -6779.741,E2 -6779.741} C_VEL
LIN {X 0,Y 481.676,Z 360.485,A -85,B 0,C 180,E1 -6782.674,E2 -6782.674} C_VEL
LIN {X 0,Y 481.64,Z 360.49,A -85,B 0,C 180,E1 -6785.709,E2 -6785.709} C_VEL
LIN {X 0,Y 481.674,Z 360.485,A -85,B 0,C 180,E1 -6788.859,E2 -6788.859} C_VEL
LIN {X 0,Y 481.655,Z 360.486,A -85,B 0,C 180,E1 -6791.913,E2 -6791.913} C_VEL
LIN {X 0,Y 481.663,Z 360.487,A -85,B 0,C 180,E1 -6794.457,E2 -6794.457} C_VEL
LIN {X 0,Y 481.65,Z 360.491,A -85,B 0,C 180,E1 -6797.839,E2 -6797.839} C_VEL
LIN {X 0,Y 481.683,Z 360.483,A -85,B 0,C 180,E1 -6800.651,E2 -6800.651} C_VEL
LIN {X 0,Y 481.63,Z 360.491,A -85,B 0,C 180,E1 -6803.376,E2 -6803.376} C_VEL
LIN {X 0,Y 481.712,Z 360.482,A -85,B 0,C 180,E1 -6806.33,E2 -6806.33} C_VEL
LIN {X 0,Y 481.653,Z 360.49,A -85,B 0,C 180,E1 -6809.417,E2 -6809.417} C_VEL
LIN {X 0,Y 481.703,Z 360.48,A -85,B 0,C 180,E1 -6812.168,E2 -6812.168} C_VEL
LIN {X 0,Y 481.721,Z 360.481,A -85,B 0,C 180,E1 -6814.97,E2 -6814.97} C_VEL
LIN {X 0,Y 481.656,Z 360.489,A -85,B 0,C 180,E1 -6817.705,E2 -6817.705} C_VEL
LIN {X 0,Y 481.711,Z 360.481,A -85,B 0,C 180,E1 -6820.393,E2 -6820.393} C_VEL
LIN {X 0,Y 481.694,Z 360.486,A -85,B 0,C 180,E1 -6823.034,E2 -6823.034} C_VEL
LIN {X 0,Y 481.693,Z 360.481,A -85,B 0,C 180,E1 -6825.639,E2 -6825.639} C_VEL
LIN {X 0,Y 481.798,Z 360.473,A -85,B 0,C 180,E1 -6828.216,E2 -6828.216} C_VEL
LIN {X 0,Y 481.766,Z 360.475,A -85,B 0,C 180,E1 -6831.612,E2 -6831.612} C_VEL
LIN {X 0,Y 481.819,Z 360.466,A -85,B 0,C 180,E1 -6834.14,E2 -6834.14} C_VEL
LIN {X 0,Y 481.93,Z 360.452,A -85,B 0,C 180,E1 -6837.492,E2 -6837.492} C_VEL
LIN {X 0,Y 481.908,Z 360.456,A -85,B 0,C 180,E1 -6840.836,E2 -6840.836} C_VEL
LIN {X 0,Y 481.931,Z 360.454,A -85,B 0,C 180,E1 -6842.507,E2 -6842.507} C_VEL
LIN {X 0,Y 481.819,Z 360.466,A -85,B 0,C 180,E1 -6845.86,E2 -6845.86} C_VEL
LIN {X 0,Y 481.765,Z 360.476,A -85,B 0,C 180,E1 -6848.388,E2 -6848.388} C_VEL
LIN {X 0,Y 481.754,Z 360.478,A -85,B 0,C 180,E1 -6851.785,E2 -6851.785} C_VEL
LIN {X 0,Y 481.745,Z 360.477,A -85,B 0,C 180,E1 -6855.224,E2 -6855.224} C_VEL
LIN {X 0,Y 481.711,Z 360.479,A -85,B 0,C 180,E1 -6858.722,E2 -6858.722} C_VEL
LIN {X 0,Y 481.648,Z 360.49,A -85,B 0,C 180,E1 -6861.395,E2 -6861.395} C_VEL
LIN {X 0,Y 481.676,Z 360.485,A -85,B 0,C 180,E1 -6864.113,E2 -6864.113} C_VEL
LIN {X 0,Y 481.749,Z 360.475,A -85,B 0,C 180,E1 -6867.139,E2 -6867.139} C_VEL
LIN {X 0,Y 481.681,Z 360.487,A -85,B 0,C 180,E1 -6869.741,E2 -6869.741} C_VEL
LIN {X 0,Y 481.674,Z 360.486,A -85,B 0,C 180,E1 -6872.674,E2 -6872.674} C_VEL
LIN {X 0,Y 481.644,Z 360.489,A -85,B 0,C 180,E1 -6875.709,E2 -6875.709} C_VEL
LIN {X 0,Y 481.673,Z 360.483,A -85,B 0,C 180,E1 -6878.859,E2 -6878.859} C_VEL
LIN {X 0,Y 481.664,Z 360.487,A -85,B 0,C 180,E1 -6881.914,E2 -6881.914} C_VEL
LIN {X 0,Y 481.662,Z 360.488,A -85,B 0,C 180,E1 -6884.457,E2 -6884.457} C_VEL
LIN {X 0,Y 481.656,Z 360.489,A -85,B 0,C 180,E1 -6887.84,E2 -6887.84} C_VEL
LIN {X 0,Y 481.663,Z 360.483,A -85,B 0,C 180,E1 -6890.654,E2 -6890.654} C_VEL
LIN {X 0,Y 481.629,Z 360.495,A -85,B 0,C 180,E1 -6893.376,E2 -6893.376} C_VEL
LIN {X 0,Y 481.712,Z 360.48,A -85,B 0,C 180,E1 -6896.33,E2 -6896.33} C_VEL
LIN {X 0,Y 481.679,Z 360.583,A -85,B 0,C 180,E1 -6897.65,E2 -6897.65} C_VEL
LIN {X 0,Y 484.235,Z 372.301,A -85,B 0,C 180,E1 -6900.432,E2 -6900.432} C_VEL
LIN {X 0,Y 484.973,Z 376.71,A -85,B 0,C 180,E1 -6901.431,E2 -6901.431} C_VEL
LIN {X 0,Y 484.109,Z 390.98,A -85,B 0,C 180,E1 -6904.412,E2 -6904.412} C_VEL
LIN {X 0,Y 483.277,Z 405.344,A -85,B 0,C 180,E1 -6907.333,E2 -6907.333} C_VEL
LIN {X 0,Y 482.613,Z 420.933,A -85,B 0,C 180,E1 -6910.431,E2 -6910.431} C_VEL
LIN {X 0,Y 481.997,Z 436.611,A -85,B 0,C 180,E1 -6913.481,E2 -6913.481} C_VEL
LIN {X 0,Y 481.788,Z 446.391,A -85,B 0,C 180,E1 -6915.318,E2 -6915.318} C_VEL
LIN {X 0,Y 483.254,Z 459.409,A -85,B 0,C 180,E1 -6915.646,E2 -6915.646} C_VEL
LIN {X 0,Y 483.329,Z 469.956,A -85,B 0,C 180,E1 -6916.011,E2 -6916.011} C_VEL
LIN {X 0,Y 482.925,Z 482.436,A -85,B 0,C 180,E1 -6916.594,E2 -6916.594} C_VEL
LIN {X 0,Y 482.569,Z 494.71,A -85,B 0,C 180,E1 -6917.362,E2 -6917.362} C_VEL
LIN {X 0,Y 482.158,Z 505.493,A -85,B 0,C 180,E1 -6918.225,E2 -6918.225} C_VEL
LIN {X 0,Y 481.796,Z 516.104,A -85,B 0,C 180,E1 -6919.281,E2 -6919.281} C_VEL
LIN {X 0,Y 481.473,Z 524.66,A -85,B 0,C 180,E1 -6920.336,E2 -6920.336} C_VEL
LIN {X 0,Y 481.264,Z 532.991,A -85,B 0,C 180,E1 -6921.603,E2 -6921.603} C_VEL
LIN {X 0,Y 481.092,Z 539.678,A -85,B 0,C 180,E1 -6922.867,E2 -6922.867} C_VEL
LIN {X 0,Y 481.019,Z 544.99,A -85,B 0,C 180,E1 -6924.13,E2 -6924.13} C_VEL
LIN {X 0,Y 480.892,Z 549.084,A -85,B 0,C 180,E1 -6925.39,E2 -6925.39} C_VEL
LIN {X 0,Y 480.963,Z 552.107,A -85,B 0,C 180,E1 -6926.649,E2 -6926.649} C_VEL
LIN {X 0,Y 480.935,Z 553.553,A -85,B 0,C 180,E1 -6927.487,E2 -6927.487} C_VEL
LIN {X 0,Y 480.809,Z 555.165,A -85,B 0,C 180,E1 -6929.163,E2 -6929.163} C_VEL
LIN {X 0,Y 480.811,Z 555.374,A -85,B 0,C 180,E1 -6930,E2 -6930} C_VEL
LIN {X 0,Y 480.812,Z 555.136,A -85,B 0,C 180,E1 -6930.838,E2 -6930.838} C_VEL
LIN {X 0,Y 480.936,Z 553.451,A -85,B 0,C 180,E1 -6932.513,E2 -6932.513} C_VEL
LIN {X 0,Y 480.978,Z 551.977,A -85,B 0,C 180,E1 -6933.351,E2 -6933.351} C_VEL
LIN {X 0,Y 480.908,Z 548.892,A -85,B 0,C 180,E1 -6934.61,E2 -6934.61} C_VEL
LIN {X 0,Y 481.039,Z 544.733,A -85,B 0,C 180,E1 -6935.87,E2 -6935.87} C_VEL
LIN {X 0,Y 481.111,Z 538.31,A -85,B 0,C 180,E1 -6937.344,E2 -6937.344} C_VEL
LIN {X 0,Y 481.285,Z 531.306,A -85,B 0,C 180,E1 -6938.608,E2 -6938.608} C_VEL
LIN {X 0,Y 481.464,Z 524.137,A -85,B 0,C 180,E1 -6939.664,E2 -6939.664} C_VEL
LIN {X 0,Y 481.749,Z 515.468,A -85,B 0,C 180,E1 -6940.72,E2 -6940.72} C_VEL
LIN {X 0,Y 482.15,Z 504.73,A -85,B 0,C 180,E1 -6941.775,E2 -6941.775} C_VEL
LIN {X 0,Y 482.494,Z 494.065,A -85,B 0,C 180,E1 -6942.62,E2 -6942.62} C_VEL
LIN {X 0,Y 482.843,Z 482.194,A -85,B 0,C 180,E1 -6943.36,E2 -6943.36} C_VEL
LIN {X 0,Y 483.223,Z 469.846,A -85,B 0,C 180,E1 -6943.939,E2 -6943.939} C_VEL
LIN {X 0,Y 483.242,Z 459.898,A -85,B 0,C 180,E1 -6944.287,E2 -6944.287} C_VEL
LIN {X 0,Y 481.9,Z 447.602,A -85,B 0,C 180,E1 -6944.611,E2 -6944.611} C_VEL
LIN {X 0,Y 481.741,Z 445.458,A -85,B 0,C 180,E1 -6944.684,E2 -6944.684} C_VEL
LIN {X 0,Y 482.215,Z 427.833,A -85,B 0,C 180,E1 -6948.042,E2 -6948.042} C_VEL
LIN {X 0,Y 482.792,Z 413.373,A -85,B 0,C 180,E1 -6950.895,E2 -6950.895} C_VEL
LIN {X 0,Y 483.675,Z 397.292,A -85,B 0,C 180,E1 -6954.235,E2 -6954.235} C_VEL
LIN {X 0,Y 484.968,Z 382.212,A -85,B 0,C 180,E1 -6957.628,E2 -6957.628} C_VEL
LIN {X 0,Y 485.295,Z 378.399,A -85,B 0,C 180,E1 -6958.549,E2 -6958.549} C_VEL
LIN {X 0,Y 484.569,Z 372.945,A -85,B 0,C 180,E1 -6960.025,E2 -6960.025} C_VEL
LIN {X 0,Y 482.757,Z 364.775,A -85,B 0,C 180,E1 -6962.592,E2 -6962.592} C_VEL
LIN {X 0,Y 481.71,Z 360.483,A -85,B 0,C 180,E1 -6964.173,E2 -6964.173} C_VEL
LIN {X 0,Y 481.633,Z 360.494,A -85,B 0,C 180,E1 -6967.797,E2 -6967.797} C_VEL
LIN {X 0,Y 481.667,Z 360.489,A -85,B 0,C 180,E1 -6970.647,E2 -6970.647} C_VEL
LIN {X 0,Y 481.669,Z 360.489,A -85,B 0,C 180,E1 -6973.297,E2 -6973.297} C_VEL
LIN {X 0,Y 481.669,Z 360.489,A -85,B 0,C 180,E1 -6976.703,E2 -6976.703} C_VEL
LIN {X 0,Y 481.694,Z 360.486,A -85,B 0,C 180,E1 -6980.061,E2 -6980.061} C_VEL
LIN {X 0,Y 481.64,Z 360.494,A -85,B 0,C 180,E1 -6982.204,E2 -6982.204} C_VEL
LIN {X 0,Y 481.695,Z 360.486,A -85,B 0,C 180,E1 -6985.318,E2 -6985.318} C_VEL
LIN {X 0,Y 481.732,Z 360.6,A -85,B 0,C 180,E1 -6987.4,E2 -6987.4} C_VEL
LIN {X 0,Y 482.235,Z 363.924,A -85,B 0,C 180,E1 -6989.331,E2 -6989.331} C_VEL
LIN {X 0,Y 482.263,Z 367.486,A -85,B 0,C 180,E1 -6991.255,E2 -6991.255} C_VEL
LIN {X 0,Y 482.038,Z 372.856,A -85,B 0,C 180,E1 -6994.062,E2 -6994.062} C_VEL
LIN {X 0,Y 481.878,Z 378.206,A -85,B 0,C 180,E1 -6996.81,E2 -6996.81} C_VEL
LIN {X 0,Y 481.675,Z 383.584,A -85,B 0,C 180,E1 -6999.502,E2 -6999.502} C_VEL
LIN {X 0,Y 481.54,Z 388.958,A -85,B 0,C 180,E1 -7002.152,E2 -7002.152} C_VEL
LIN {X 0,Y 481.435,Z 394.321,A -85,B 0,C 180,E1 -7004.766,E2 -7004.766} C_VEL
LIN {X 0,Y 481.299,Z 401.495,A -85,B 0,C 180,E1 -7008.204,E2 -7008.204} C_VEL
LIN {X 0,Y 481.188,Z 407.597,A -85,B 0,C 180,E1 -7011.006,E2 -7011.006} C_VEL
LIN {X 0,Y 482.424,Z 415.899,A -85,B 0,C 180,E1 -7011.412,E2 -7011.412} C_VEL
LIN {X 0,Y 482.245,Z 425.14,A -85,B 0,C 180,E1 -7011.968,E2 -7011.968} C_VEL
LIN {X 0,Y 482.091,Z 433.362,A -85,B 0,C 180,E1 -7012.625,E2 -7012.625} C_VEL
LIN {X 0,Y 481.841,Z 440.032,A -85,B 0,C 180,E1 -7013.299,E2 -7013.299} C_VEL
LIN {X 0,Y 481.595,Z 446.617,A -85,B 0,C 180,E1 -7014.137,E2 -7014.137} C_VEL
LIN {X 0,Y 481.453,Z 451.826,A -85,B 0,C 180,E1 -7014.975,E2 -7014.975} C_VEL
LIN {X 0,Y 481.341,Z 455.914,A -85,B 0,C 180,E1 -7015.813,E2 -7015.813} C_VEL
LIN {X 0,Y 481.204,Z 459.105,A -85,B 0,C 180,E1 -7016.651,E2 -7016.651} C_VEL
LIN {X 0,Y 481.045,Z 461.499,A -85,B 0,C 180,E1 -7017.488,E2 -7017.488} C_VEL
LIN {X 0,Y 480.956,Z 463.153,A -85,B 0,C 180,E1 -7018.325,E2 -7018.325} C_VEL
LIN {X 0,Y 480.921,Z 464.112,A -85,B 0,C 180,E1 -7019.163,E2 -7019.163} C_VEL
LIN {X 0,Y 480.907,Z 464.403,A -85,B 0,C 180,E1 -7020,E2 -7020} C_VEL
LIN {X 0,Y 480.904,Z 464.03,A -85,B 0,C 180,E1 -7020.837,E2 -7020.837} C_VEL
LIN {X 0,Y 480.925,Z 462.989,A -85,B 0,C 180,E1 -7021.675,E2 -7021.675} C_VEL
LIN {X 0,Y 481.008,Z 461.255,A -85,B 0,C 180,E1 -7022.512,E2 -7022.512} C_VEL
LIN {X 0,Y 481.187,Z 458.775,A -85,B 0,C 180,E1 -7023.349,E2 -7023.349} C_VEL
LIN {X 0,Y 481.335,Z 455.48,A -85,B 0,C 180,E1 -7024.187,E2 -7024.187} C_VEL
LIN {X 0,Y 481.449,Z 450.065,A -85,B 0,C 180,E1 -7025.235,E2 -7025.235} C_VEL
LIN {X 0,Y 481.545,Z 444.451,A -85,B 0,C 180,E1 -7026.074,E2 -7026.074} C_VEL
LIN {X 0,Y 481.666,Z 437.978,A -85,B 0,C 180,E1 -7026.841,E2 -7026.841} C_VEL
LIN {X 0,Y 481.897,Z 429.216,A -85,B 0,C 180,E1 -7027.648,E2 -7027.648} C_VEL
LIN {X 0,Y 482.143,Z 420.113,A -85,B 0,C 180,E1 -7028.276,E2 -7028.276} C_VEL
LIN {X 0,Y 482.08,Z 413.173,A -85,B 0,C 180,E1 -7028.647,E2 -7028.647} C_VEL
LIN {X 0,Y 481.008,Z 405.903,A -85,B 0,C 180,E1 -7028.984,E2 -7028.984} C_VEL
LIN {X 0,Y 481.065,Z 399.684,A -85,B 0,C 180,E1 -7031.812,E2 -7031.812} C_VEL
LIN {X 0,Y 481.215,Z 391.799,A -85,B 0,C 180,E1 -7035.439,E2 -7035.439} C_VEL
LIN {X 0,Y 481.284,Z 384.715,A -85,B 0,C 180,E1 -7038.739,E2 -7038.739} C_VEL
LIN {X 0,Y 481.366,Z 379.075,A -85,B 0,C 180,E1 -7041.408,E2 -7041.408} C_VEL
LIN {X 0,Y 481.472,Z 373.375,A -85,B 0,C 180,E1 -7044.124,E2 -7044.124} C_VEL
LIN {X 0,Y 481.654,Z 367.193,A -85,B 0,C 180,E1 -7047.117,E2 -7047.117} C_VEL
LIN {X 0,Y 481.872,Z 360.925,A -85,B 0,C 180,E1 -7050.163,E2 -7050.163} C_VEL
LIN {X 0,Y 481.787,Z 360.474,A -85,B 0,C 180,E1 -7050.53,E2 -7050.53} C_VEL
LIN {X 0,Y 481.7,Z 360.48,A -85,B 0,C 180,E1 -7053.733,E2 -7053.733} C_VEL
LIN {X 0,Y 481.632,Z 360.491,A -85,B 0,C 180,E1 -7056.747,E2 -7056.747} C_VEL
LIN {X 0,Y 481.68,Z 360.486,A -85,B 0,C 180,E1 -7059.94,E2 -7059.94} C_VEL
LIN {X 0,Y 481.642,Z 360.488,A -85,B 0,C 180,E1 -7063.3,E2 -7063.3} C_VEL
LIN {X 0,Y 481.663,Z 360.486,A -85,B 0,C 180,E1 -7065.641,E2 -7065.641} C_VEL
LIN {X 0,Y 481.666,Z 360.486,A -85,B 0,C 180,E1 -7068.959,E2 -7068.959} C_VEL
LIN {X 0,Y 481.658,Z 360.487,A -85,B 0,C 180,E1 -7071.993,E2 -7071.993} C_VEL
LIN {X 0,Y 481.692,Z 360.481,A -85,B 0,C 180,E1 -7075.318,E2 -7075.318} C_VEL
LIN {X 0,Y 481.649,Z 360.49,A -85,B 0,C 180,E1 -7078.312,E2 -7078.312} C_VEL
LIN {X 0,Y 481.704,Z 360.483,A -85,B 0,C 180,E1 -7081.219,E2 -7081.219} C_VEL
LIN {X 0,Y 481.693,Z 360.482,A -85,B 0,C 180,E1 -7084.042,E2 -7084.042} C_VEL
LIN {X 0,Y 481.654,Z 360.486,A -85,B 0,C 180,E1 -7087.155,E2 -7087.155} C_VEL
LIN {X 0,Y 480.972,Z 360.575,A -85,B 0,C 180,E1 -7087.853,E2 -7087.853} C_VEL
LIN {X 0,Y 478.116,Z 360.928,A -85,B 0,C 180,E1 -7088.987,E2 -7088.987} C_VEL
LIN {X 0,Y 475.728,Z 361.229,A -85,B 0,C 180,E1 -7089.901,E2 -7089.901} C_VEL
LIN {X 0,Y 474.728,Z 361.351,A -85,B 0,C 180,E1 -7090.607,E2 -7090.607} C_VEL
LIN {X 0,Y 474.659,Z 361.36,A -85,B 0,C 180,E1 -7090.846,E2 -7090.846} C_VEL
LIN {X 0,Y 474.685,Z 361.357,A -85,B 0,C 180,E1 -7094.232,E2 -7094.232} C_VEL
LIN {X 0,Y 474.705,Z 361.353,A -85,B 0,C 180,E1 -7097.724,E2 -7097.724} C_VEL
LIN {X 0,Y 474.707,Z 361.353,A -85,B 0,C 180,E1 -7100.627,E2 -7100.627} C_VEL
LIN {X 0,Y 474.743,Z 361.35,A -85,B 0,C 180,E1 -7103.198,E2 -7103.198} C_VEL
LIN {X 0,Y 474.621,Z 361.363,A -85,B 0,C 180,E1 -7105.754,E2 -7105.754} C_VEL
LIN {X 0,Y 474.898,Z 361.328,A -85,B 0,C 180,E1 -7107.455,E2 -7107.455} C_VEL
LIN {X 0,Y 474.916,Z 361.329,A -85,B 0,C 180,E1 -7110,E2 -7110} C_VEL
LIN {X 0,Y 474.898,Z 361.33,A -85,B 0,C 180,E1 -7112.545,E2 -7112.545} C_VEL
LIN {X 0,Y 474.775,Z 361.346,A -85,B 0,C 180,E1 -7115.948,E2 -7115.948} C_VEL
LIN {X 0,Y 474.732,Z 361.348,A -85,B 0,C 180,E1 -7118.513,E2 -7118.513} C_VEL
LIN {X 0,Y 474.708,Z 361.353,A -85,B 0,C 180,E1 -7121.962,E2 -7121.962} C_VEL
LIN {X 0,Y 474.704,Z 361.353,A -85,B 0,C 180,E1 -7125.456,E2 -7125.456} C_VEL
LIN {X 0,Y 474.67,Z 361.356,A -85,B 0,C 180,E1 -7129.01,E2 -7129.01} C_VEL
LIN {X 0,Y 474.592,Z 361.368,A -85,B 0,C 180,E1 -7131.729,E2 -7131.729} C_VEL
LIN {X 0,Y 474.661,Z 361.36,A -85,B 0,C 180,E1 -7134.493,E2 -7134.493} C_VEL
LIN {X 0,Y 474.703,Z 361.354,A -85,B 0,C 180,E1 -7137.339,E2 -7137.339} C_VEL
LIN {X 0,Y 474.608,Z 361.364,A -85,B 0,C 180,E1 -7140.81,E2 -7140.81} C_VEL
LIN {X 0,Y 474.64,Z 361.361,A -85,B 0,C 180,E1 -7143.984,E2 -7143.984} C_VEL
LIN {X 0,Y 474.575,Z 361.37,A -85,B 0,C 180,E1 -7146.899,E2 -7146.899} C_VEL
LIN {X 0,Y 474.631,Z 361.366,A -85,B 0,C 180,E1 -7149.648,E2 -7149.648} C_VEL
LIN {X 0,Y 474.634,Z 361.364,A -85,B 0,C 180,E1 -7152.932,E2 -7152.932} C_VEL
LIN {X 0,Y 474.612,Z 361.366,A -85,B 0,C 180,E1 -7155.895,E2 -7155.895} C_VEL
LIN {X 0,Y 474.63,Z 361.363,A -85,B 0,C 180,E1 -7159.041,E2 -7159.041} C_VEL
LIN {X 0,Y 474.612,Z 361.365,A -85,B 0,C 180,E1 -7161.704,E2 -7161.704} C_VEL
LIN {X 0,Y 474.627,Z 361.366,A -85,B 0,C 180,E1 -7164.726,E2 -7164.726} C_VEL
LIN {X 0,Y 474.638,Z 361.364,A -85,B 0,C 180,E1 -7167.788,E2 -7167.788} C_VEL
LIN {X 0,Y 474.627,Z 361.363,A -85,B 0,C 180,E1 -7170.884,E2 -7170.884} C_VEL
LIN {X 0,Y 474.663,Z 361.357,A -85,B 0,C 180,E1 -7173.628,E2 -7173.628} C_VEL
LIN {X 0,Y 474.639,Z 361.365,A -85,B 0,C 180,E1 -7176.641,E2 -7176.641} C_VEL
LIN {X 0,Y 474.66,Z 361.361,A -85,B 0,C 180,E1 -7180.09,E2 -7180.09} C_VEL
LIN {X 0,Y 474.653,Z 361.361,A -85,B 0,C 180,E1 -7182.774,E2 -7182.774} C_VEL
LIN {X 0,Y 474.651,Z 361.358,A -85,B 0,C 180,E1 -7185.421,E2 -7185.421} C_VEL
LIN {X 0,Y 474.742,Z 361.35,A -85,B 0,C 180,E1 -7188.038,E2 -7188.038} C_VEL
LIN {X 0,Y 474.731,Z 361.351,A -85,B 0,C 180,E1 -7191.486,E2 -7191.486} C_VEL
LIN {X 0,Y 474.782,Z 361.343,A -85,B 0,C 180,E1 -7194.052,E2 -7194.052} C_VEL
LIN {X 0,Y 474.896,Z 361.328,A -85,B 0,C 180,E1 -7197.455,E2 -7197.455} C_VEL
LIN {X 0,Y 474.915,Z 361.33,A -85,B 0,C 180,E1 -7200,E2 -7200} C_VEL
LIN {X 0,Y 474.897,Z 361.33,A -85,B 0,C 180,E1 -7202.545,E2 -7202.545} C_VEL
LIN {X 0,Y 474.781,Z 361.343,A -85,B 0,C 180,E1 -7205.948,E2 -7205.948} C_VEL
LIN {X 0,Y 474.73,Z 361.351,A -85,B 0,C 180,E1 -7208.513,E2 -7208.513} C_VEL
LIN {X 0,Y 474.707,Z 361.354,A -85,B 0,C 180,E1 -7211.962,E2 -7211.962} C_VEL
LIN {X 0,Y 474.702,Z 361.353,A -85,B 0,C 180,E1 -7215.456,E2 -7215.456} C_VEL
LIN {X 0,Y 474.666,Z 361.357,A -85,B 0,C 180,E1 -7219.01,E2 -7219.01} C_VEL
LIN {X 0,Y 474.591,Z 361.37,A -85,B 0,C 180,E1 -7221.729,E2 -7221.729} C_VEL
LIN {X 0,Y 474.659,Z 361.361,A -85,B 0,C 180,E1 -7224.493,E2 -7224.493} C_VEL
LIN {X 0,Y 474.683,Z 361.355,A -85,B 0,C 180,E1 -7227.334,E2 -7227.334} C_VEL
LIN {X 0,Y 474.607,Z 361.366,A -85,B 0,C 180,E1 -7230.23,E2 -7230.23} C_VEL
LIN {X 0,Y 474.645,Z 361.363,A -85,B 0,C 180,E1 -7233.22,E2 -7233.22} C_VEL
LIN {X 0,Y 474.595,Z 361.37,A -85,B 0,C 180,E1 -7236.323,E2 -7236.323} C_VEL
LIN {X 0,Y 474.63,Z 361.365,A -85,B 0,C 180,E1 -7239.648,E2 -7239.648} C_VEL
LIN {X 0,Y 474.637,Z 361.363,A -85,B 0,C 180,E1 -7242.932,E2 -7242.932} C_VEL
LIN {X 0,Y 474.617,Z 361.365,A -85,B 0,C 180,E1 -7245.896,E2 -7245.896} C_VEL
LIN {X 0,Y 474.634,Z 361.361,A -85,B 0,C 180,E1 -7249.04,E2 -7249.04} C_VEL
LIN {X 0,Y 474.612,Z 361.367,A -85,B 0,C 180,E1 -7251.704,E2 -7251.704} C_VEL
LIN {X 0,Y 474.626,Z 361.366,A -85,B 0,C 180,E1 -7254.726,E2 -7254.726} C_VEL
LIN {X 0,Y 474.629,Z 361.359,A -85,B 0,C 180,E1 -7257.32,E2 -7257.32} C_VEL
LIN {X 0,Y 476.962,Z 372.132,A -85,B 0,C 180,E1 -7259.935,E2 -7259.935} C_VEL
LIN {X 0,Y 478.023,Z 377.621,A -85,B 0,C 180,E1 -7261.217,E2 -7261.217} C_VEL
LIN {X 0,Y 477.502,Z 386.382,A -85,B 0,C 180,E1 -7263.09,E2 -7263.09} C_VEL
LIN {X 0,Y 476.594,Z 401.305,A -85,B 0,C 180,E1 -7266.21,E2 -7266.21} C_VEL
LIN {X 0,Y 475.747,Z 417.252,A -85,B 0,C 180,E1 -7269.461,E2 -7269.461} C_VEL
LIN {X 0,Y 475.08,Z 433.935,A -85,B 0,C 180,E1 -7272.791,E2 -7272.791} C_VEL
LIN {X 0,Y 474.696,Z 445.923,A -85,B 0,C 180,E1 -7275.135,E2 -7275.135} C_VEL
LIN {X 0,Y 476.16,Z 459.433,A -85,B 0,C 180,E1 -7275.482,E2 -7275.482} C_VEL
LIN {X 0,Y 476.413,Z 463.398,A -85,B 0,C 180,E1 -7275.613,E2 -7275.613} C_VEL
LIN {X 0,Y 476.155,Z 475.923,A -85,B 0,C 180,E1 -7276.122,E2 -7276.122} C_VEL
LIN {X 0,Y 475.778,Z 487.623,A -85,B 0,C 180,E1 -7276.764,E2 -7276.764} C_VEL
LIN {X 0,Y 475.424,Z 499.147,A -85,B 0,C 180,E1 -7277.585,E2 -7277.585} C_VEL
LIN {X 0,Y 474.939,Z 510.234,A -85,B 0,C 180,E1 -7278.585,E2 -7278.585} C_VEL
LIN {X 0,Y 474.599,Z 518.918,A -85,B 0,C 180,E1 -7279.549,E2 -7279.549} C_VEL
LIN {X 0,Y 474.339,Z 526.906,A -85,B 0,C 180,E1 -7280.62,E2 -7280.62} C_VEL
LIN {X 0,Y 474.1,Z 534.669,A -85,B 0,C 180,E1 -7281.904,E2 -7281.904} C_VEL
LIN {X 0,Y 473.976,Z 540.88,A -85,B 0,C 180,E1 -7283.187,E2 -7283.187} C_VEL
LIN {X 0,Y 473.938,Z 545.786,A -85,B 0,C 180,E1 -7284.469,E2 -7284.469} C_VEL
LIN {X 0,Y 473.875,Z 549.523,A -85,B 0,C 180,E1 -7285.747,E2 -7285.747} C_VEL
LIN {X 0,Y 473.889,Z 551.444,A -85,B 0,C 180,E1 -7286.599,E2 -7286.599} C_VEL
LIN {X 0,Y 473.876,Z 552.897,A -85,B 0,C 180,E1 -7287.45,E2 -7287.45} C_VEL
LIN {X 0,Y 473.739,Z 554.507,A -85,B 0,C 180,E1 -7289.15,E2 -7289.15} C_VEL
LIN {X 0,Y 473.742,Z 554.715,A -85,B 0,C 180,E1 -7290,E2 -7290} C_VEL
LIN {X 0,Y 473.742,Z 554.471,A -85,B 0,C 180,E1 -7290.85,E2 -7290.85} C_VEL
LIN {X 0,Y 473.878,Z 552.775,A -85,B 0,C 180,E1 -7292.55,E2 -7292.55} C_VEL
LIN {X 0,Y 473.904,Z 551.289,A -85,B 0,C 180,E1 -7293.401,E2 -7293.401} C_VEL
LIN {X 0,Y 473.823,Z 548.184,A -85,B 0,C 180,E1 -7294.679,E2 -7294.679} C_VEL
LIN {X 0,Y 473.948,Z 543.998,A -85,B 0,C 180,E1 -7295.958,E2 -7295.958} C_VEL
LIN {X 0,Y 474.023,Z 537.544,A -85,B 0,C 180,E1 -7297.454,E2 -7297.454} C_VEL
LIN {X 0,Y 474.184,Z 530.505,A -85,B 0,C 180,E1 -7298.738,E2 -7298.738} C_VEL
LIN {X 0,Y 474.41,Z 523.303,A -85,B 0,C 180,E1 -7299.809,E2 -7299.809} C_VEL
LIN {X 0,Y 474.728,Z 514.569,A -85,B 0,C 180,E1 -7300.88,E2 -7300.88} C_VEL
LIN {X 0,Y 475.095,Z 504.955,A -85,B 0,C 180,E1 -7301.844,E2 -7301.844} C_VEL
LIN {X 0,Y 475.43,Z 494.878,A -85,B 0,C 180,E1 -7302.672,E2 -7302.672} C_VEL
LIN {X 0,Y 475.81,Z 482.97,A -85,B 0,C 180,E1 -7303.452,E2 -7303.452} C_VEL
LIN {X 0,Y 476.235,Z 471.093,A -85,B 0,C 180,E1 -7304.039,E2 -7304.039} C_VEL
LIN {X 0,Y 476.311,Z 460.987,A -85,B 0,C 180,E1 -7304.418,E2 -7304.418} C_VEL
LIN {X 0,Y 474.972,Z 448.308,A -85,B 0,C 180,E1 -7304.774,E2 -7304.774} C_VEL
LIN {X 0,Y 474.657,Z 445.221,A -85,B 0,C 180,E1 -7304.853,E2 -7304.853} C_VEL
LIN {X 0,Y 475.183,Z 428.582,A -85,B 0,C 180,E1 -7308.095,E2 -7308.095} C_VEL
LIN {X 0,Y 475.834,Z 413.498,A -85,B 0,C 180,E1 -7311.138,E2 -7311.138} C_VEL
LIN {X 0,Y 476.776,Z 398.379,A -85,B 0,C 180,E1 -7314.377,E2 -7314.377} C_VEL
LIN {X 0,Y 478.049,Z 384.435,A -85,B 0,C 180,E1 -7317.587,E2 -7317.587} C_VEL
LIN {X 0,Y 478.409,Z 378.808,A -85,B 0,C 180,E1 -7318.998,E2 -7318.998} C_VEL
LIN {X 0,Y 477.481,Z 373.537,A -85,B 0,C 180,E1 -7320.518,E2 -7320.518} C_VEL
LIN {X 0,Y 475.686,Z 365.706,A -85,B 0,C 180,E1 -7323.138,E2 -7323.138} C_VEL
LIN {X 0,Y 474.636,Z 361.366,A -85,B 0,C 180,E1 -7324.885,E2 -7324.885} C_VEL
LIN {X 0,Y 474.614,Z 361.368,A -85,B 0,C 180,E1 -7328.457,E2 -7328.457} C_VEL
LIN {X 0,Y 474.635,Z 361.365,A -85,B 0,C 180,E1 -7330.96,E2 -7330.96} C_VEL
LIN {X 0,Y 474.618,Z 361.367,A -85,B 0,C 180,E1 -7334.104,E2 -7334.104} C_VEL
LIN {X 0,Y 474.638,Z 361.364,A -85,B 0,C 180,E1 -7337.068,E2 -7337.068} C_VEL
LIN {X 0,Y 474.675,Z 361.36,A -85,B 0,C 180,E1 -7340.457,E2 -7340.457} C_VEL
LIN {X 0,Y 474.595,Z 361.371,A -85,B 0,C 180,E1 -7343.677,E2 -7343.677} C_VEL
LIN {X 0,Y 474.677,Z 361.471,A -85,B 0,C 180,E1 -7346.888,E2 -7346.888} C_VEL
LIN {X 0,Y 475.234,Z 365.047,A -85,B 0,C 180,E1 -7349.064,E2 -7349.064} C_VEL
LIN {X 0,Y 475.331,Z 368.137,A -85,B 0,C 180,E1 -7350.796,E2 -7350.796} C_VEL
LIN {X 0,Y 475.103,Z 373.446,A -85,B 0,C 180,E1 -7353.655,E2 -7353.655} C_VEL
LIN {X 0,Y 474.877,Z 379.024,A -85,B 0,C 180,E1 -7356.575,E2 -7356.575} C_VEL
LIN {X 0,Y 474.7,Z 384.097,A -85,B 0,C 180,E1 -7359.187,E2 -7359.187} C_VEL
LIN {X 0,Y 474.566,Z 389.483,A -85,B 0,C 180,E1 -7361.881,E2 -7361.881} C_VEL
LIN {X 0,Y 474.426,Z 394.861,A -85,B 0,C 180,E1 -7364.535,E2 -7364.535} C_VEL
LIN {X 0,Y 474.258,Z 402.045,A -85,B 0,C 180,E1 -7368.026,E2 -7368.026} C_VEL
LIN {X 0,Y 474.13,Z 407.95,A -85,B 0,C 180,E1 -7370.804,E2 -7370.804} C_VEL
LIN {X 0,Y 475.457,Z 415.433,A -85,B 0,C 180,E1 -7371.178,E2 -7371.178} C_VEL
LIN {X 0,Y 475.359,Z 424.697,A -85,B 0,C 180,E1 -7371.733,E2 -7371.733} C_VEL
LIN {X 0,Y 475.148,Z 433.583,A -85,B 0,C 180,E1 -7372.443,E2 -7372.443} C_VEL
LIN {X 0,Y 474.855,Z 440.935,A -85,B 0,C 180,E1 -7373.2,E2 -7373.2} C_VEL
LIN {X 0,Y 474.596,Z 447.434,A -85,B 0,C 180,E1 -7374.05,E2 -7374.05} C_VEL
LIN {X 0,Y 474.415,Z 453.691,A -85,B 0,C 180,E1 -7375.114,E2 -7375.114} C_VEL
LIN {X 0,Y 474.358,Z 458.341,A -85,B 0,C 180,E1 -7376.177,E2 -7376.177} C_VEL
LIN {X 0,Y 473.99,Z 462.221,A -85,B 0,C 180,E1 -7377.451,E2 -7377.451} C_VEL
LIN {X 0,Y 473.896,Z 463.863,A -85,B 0,C 180,E1 -7378.3,E2 -7378.3} C_VEL
LIN {X 0,Y 473.857,Z 464.81,A -85,B 0,C 180,E1 -7379.15,E2 -7379.15} C_VEL
LIN {X 0,Y 473.841,Z 465.087,A -85,B 0,C 180,E1 -7380,E2 -7380} C_VEL
LIN {X 0,Y 473.837,Z 464.698,A -85,B 0,C 180,E1 -7380.85,E2 -7380.85} C_VEL
LIN {X 0,Y 473.859,Z 463.639,A -85,B 0,C 180,E1 -7381.7,E2 -7381.7} C_VEL
LIN {X 0,Y 473.952,Z 461.886,A -85,B 0,C 180,E1 -7382.55,E2 -7382.55} C_VEL
LIN {X 0,Y 474.143,Z 459.386,A -85,B 0,C 180,E1 -7383.399,E2 -7383.399} C_VEL
LIN {X 0,Y 474.307,Z 456.072,A -85,B 0,C 180,E1 -7384.249,E2 -7384.249} C_VEL
LIN {X 0,Y 474.425,Z 450.632,A -85,B 0,C 180,E1 -7385.312,E2 -7385.312} C_VEL
LIN {X 0,Y 474.528,Z 444.997,A -85,B 0,C 180,E1 -7386.164,E2 -7386.164} C_VEL
LIN {X 0,Y 474.649,Z 438.465,A -85,B 0,C 180,E1 -7386.948,E2 -7386.948} C_VEL
LIN {X 0,Y 474.88,Z 429.76,A -85,B 0,C 180,E1 -7387.761,E2 -7387.761} C_VEL
LIN {X 0,Y 475.152,Z 420.694,A -85,B 0,C 180,E1 -7388.399,E2 -7388.399} C_VEL
LIN {X 0,Y 475.075,Z 413.824,A -85,B 0,C 180,E1 -7388.775,E2 -7388.775} C_VEL
LIN {X 0,Y 473.934,Z 406.215,A -85,B 0,C 180,E1 -7389.119,E2 -7389.119} C_VEL
LIN {X 0,Y 474,Z 399.963,A -85,B 0,C 180,E1 -7391.981,E2 -7391.981} C_VEL
LIN {X 0,Y 474.153,Z 392.288,A -85,B 0,C 180,E1 -7395.539,E2 -7395.539} C_VEL
LIN {X 0,Y 474.232,Z 384.874,A -85,B 0,C 180,E1 -7399.028,E2 -7399.028} C_VEL
LIN {X 0,Y 474.325,Z 379.193,A -85,B 0,C 180,E1 -7401.742,E2 -7401.742} C_VEL
LIN {X 0,Y 474.455,Z 373.468,A -85,B 0,C 180,E1 -7404.504,E2 -7404.504} C_VEL
LIN {X 0,Y 474.605,Z 367.653,A -85,B 0,C 180,E1 -7407.326,E2 -7407.326} C_VEL
LIN {X 0,Y 474.772,Z 361.389,A -85,B 0,C 180,E1 -7410.421,E2 -7410.421} C_VEL
LIN {X 0,Y 474.642,Z 361.36,A -85,B 0,C 180,E1 -7413.984,E2 -7413.984} C_VEL
LIN {X 0,Y 474.578,Z 361.369,A -85,B 0,C 180,E1 -7416.9,E2 -7416.9} C_VEL
LIN {X 0,Y 474.631,Z 361.364,A -85,B 0,C 180,E1 -7419.648,E2 -7419.648} C_VEL
LIN {X 0,Y 474.618,Z 361.368,A -85,B 0,C 180,E1 -7422.934,E2 -7422.934} C_VEL
LIN {X 0,Y 474.619,Z 361.364,A -85,B 0,C 180,E1 -7425.896,E2 -7425.896} C_VEL
LIN {X 0,Y 474.636,Z 361.363,A -85,B 0,C 180,E1 -7429.04,E2 -7429.04} C_VEL
LIN {X 0,Y 474.613,Z 361.365,A -85,B 0,C 180,E1 -7431.704,E2 -7431.704} C_VEL
LIN {X 0,Y 474.628,Z 361.366,A -85,B 0,C 180,E1 -7434.726,E2 -7434.726} C_VEL
LIN {X 0,Y 474.64,Z 361.362,A -85,B 0,C 180,E1 -7437.788,E2 -7437.788} C_VEL
LIN {X 0,Y 474.628,Z 361.365,A -85,B 0,C 180,E1 -7440.884,E2 -7440.884} C_VEL
LIN {X 0,Y 474.658,Z 361.358,A -85,B 0,C 180,E1 -7443.628,E2 -7443.628} C_VEL
LIN {X 0,Y 474.638,Z 361.362,A -85,B 0,C 180,E1 -7446.642,E2 -7446.642} C_VEL
LIN {X 0,Y 474.659,Z 361.36,A -85,B 0,C 180,E1 -7450.09,E2 -7450.09} C_VEL
LIN {X 0,Y 474.659,Z 361.36,A -85,B 0,C 180,E1 -7450.846,E2 -7450.846} C_VEL
LIN {X 0,Y 474.031,Z 361.442,A -85,B 0,C 180,E1 -7451.554,E2 -7451.554} C_VEL
LIN {X 0,Y 471.202,Z 361.797,A -85,B 0,C 180,E1 -7452.704,E2 -7452.704} C_VEL
LIN {X 0,Y 468.776,Z 362.096,A -85,B 0,C 180,E1 -7453.631,E2 -7453.631} C_VEL
LIN {X 0,Y 467.715,Z 362.226,A -85,B 0,C 180,E1 -7454.347,E2 -7454.347} C_VEL
LIN {X 0,Y 467.621,Z 362.235,A -85,B 0,C 180,E1 -7454.589,E2 -7454.589} C_VEL
LIN {X 0,Y 467.66,Z 362.232,A -85,B 0,C 180,E1 -7457.855,E2 -7457.855} C_VEL
LIN {X 0,Y 467.685,Z 362.229,A -85,B 0,C 180,E1 -7461.357,E2 -7461.357} C_VEL
LIN {X 0,Y 467.74,Z 362.221,A -85,B 0,C 180,E1 -7463.962,E2 -7463.962} C_VEL
LIN {X 0,Y 467.863,Z 362.204,A -85,B 0,C 180,E1 -7467.417,E2 -7467.417} C_VEL
LIN {X 0,Y 467.887,Z 362.204,A -85,B 0,C 180,E1 -7470,E2 -7470} C_VEL
LIN {X 0,Y 467.863,Z 362.207,A -85,B 0,C 180,E1 -7472.583,E2 -7472.583} C_VEL
LIN {X 0,Y 467.739,Z 362.223,A -85,B 0,C 180,E1 -7476.037,E2 -7476.037} C_VEL
LIN {X 0,Y 467.685,Z 362.225,A -85,B 0,C 180,E1 -7478.643,E2 -7478.643} C_VEL
LIN {X 0,Y 467.66,Z 362.231,A -85,B 0,C 180,E1 -7482.145,E2 -7482.145} C_VEL
LIN {X 0,Y 467.643,Z 362.233,A -85,B 0,C 180,E1 -7485.695,E2 -7485.695} C_VEL
LIN {X 0,Y 467.622,Z 362.234,A -85,B 0,C 180,E1 -7488.765,E2 -7488.765} C_VEL
LIN {X 0,Y 467.584,Z 362.242,A -85,B 0,C 180,E1 -7491.268,E2 -7491.268} C_VEL
LIN {X 0,Y 467.575,Z 362.241,A -85,B 0,C 180,E1 -7493.943,E2 -7493.943} C_VEL
LIN {X 0,Y 467.62,Z 362.237,A -85,B 0,C 180,E1 -7496.8,E2 -7496.8} C_VEL
LIN {X 0,Y 467.557,Z 362.246,A -85,B 0,C 180,E1 -7499.738,E2 -7499.738} C_VEL
LIN {X 0,Y 467.586,Z 362.24,A -85,B 0,C 180,E1 -7502.758,E2 -7502.758} C_VEL
LIN {X 0,Y 467.556,Z 362.245,A -85,B 0,C 180,E1 -7505.889,E2 -7505.889} C_VEL
LIN {X 0,Y 467.585,Z 362.24,A -85,B 0,C 180,E1 -7509.145,E2 -7509.145} C_VEL
LIN {X 0,Y 467.589,Z 362.238,A -85,B 0,C 180,E1 -7512.567,E2 -7512.567} C_VEL
LIN {X 0,Y 467.573,Z 362.244,A -85,B 0,C 180,E1 -7515.053,E2 -7515.053} C_VEL
LIN {X 0,Y 467.591,Z 362.24,A -85,B 0,C 180,E1 -7517.44,E2 -7517.44} C_VEL
LIN {X 0,Y 467.585,Z 362.24,A -85,B 0,C 180,E1 -7520.855,E2 -7520.855} C_VEL
LIN {X 0,Y 467.562,Z 362.242,A -85,B 0,C 180,E1 -7524.261,E2 -7524.261} C_VEL
LIN {X 0,Y 467.584,Z 362.24,A -85,B 0,C 180,E1 -7527.321,E2 -7527.321} C_VEL
LIN {X 0,Y 467.573,Z 362.242,A -85,B 0,C 180,E1 -7530.667,E2 -7530.667} C_VEL
LIN {X 0,Y 467.619,Z 362.238,A -85,B 0,C 180,E1 -7533.2,E2 -7533.2} C_VEL
LIN {X 0,Y 467.596,Z 362.241,A -85,B 0,C 180,E1 -7536.468,E2 -7536.468} C_VEL
LIN {X 0,Y 467.627,Z 362.236,A -85,B 0,C 180,E1 -7539.777,E2 -7539.777} C_VEL
LIN {X 0,Y 467.612,Z 362.237,A -85,B 0,C 180,E1 -7542.507,E2 -7542.507} C_VEL
LIN {X 0,Y 467.609,Z 362.237,A -85,B 0,C 180,E1 -7545.196,E2 -7545.196} C_VEL
LIN {X 0,Y 467.686,Z 362.228,A -85,B 0,C 180,E1 -7547.855,E2 -7547.855} C_VEL
LIN {X 0,Y 467.685,Z 362.229,A -85,B 0,C 180,E1 -7551.357,E2 -7551.357} C_VEL
LIN {X 0,Y 467.746,Z 362.219,A -85,B 0,C 180,E1 -7553.963,E2 -7553.963} C_VEL
LIN {X 0,Y 467.862,Z 362.205,A -85,B 0,C 180,E1 -7557.417,E2 -7557.417} C_VEL
LIN {X 0,Y 467.886,Z 362.206,A -85,B 0,C 180,E1 -7560,E2 -7560} C_VEL
LIN {X 0,Y 467.862,Z 362.207,A -85,B 0,C 180,E1 -7562.583,E2 -7562.583} C_VEL
LIN {X 0,Y 467.746,Z 362.22,A -85,B 0,C 180,E1 -7566.037,E2 -7566.037} C_VEL
LIN {X 0,Y 467.683,Z 362.228,A -85,B 0,C 180,E1 -7568.643,E2 -7568.643} C_VEL
LIN {X 0,Y 467.659,Z 362.231,A -85,B 0,C 180,E1 -7572.145,E2 -7572.145} C_VEL
LIN {X 0,Y 467.641,Z 362.232,A -85,B 0,C 180,E1 -7575.695,E2 -7575.695} C_VEL
LIN {X 0,Y 467.625,Z 362.234,A -85,B 0,C 180,E1 -7579.308,E2 -7579.308} C_VEL
LIN {X 0,Y 467.537,Z 362.247,A -85,B 0,C 180,E1 -7582.074,E2 -7582.074} C_VEL
LIN {X 0,Y 467.605,Z 362.239,A -85,B 0,C 180,E1 -7584.887,E2 -7584.887} C_VEL
LIN {X 0,Y 467.622,Z 362.236,A -85,B 0,C 180,E1 -7587.769,E2 -7587.769} C_VEL
LIN {X 0,Y 467.57,Z 362.242,A -85,B 0,C 180,E1 -7591.045,E2 -7591.045} C_VEL
LIN {X 0,Y 467.592,Z 362.24,A -85,B 0,C 180,E1 -7594.243,E2 -7594.243} C_VEL
LIN {X 0,Y 467.553,Z 362.244,A -85,B 0,C 180,E1 -7597.187,E2 -7597.187} C_VEL
LIN {X 0,Y 467.581,Z 362.24,A -85,B 0,C 180,E1 -7600.264,E2 -7600.264} C_VEL
LIN {X 0,Y 467.588,Z 362.24,A -85,B 0,C 180,E1 -7602.567,E2 -7602.567} C_VEL
LIN {X 0,Y 467.573,Z 362.244,A -85,B 0,C 180,E1 -7605.053,E2 -7605.053} C_VEL
LIN {X 0,Y 467.591,Z 362.239,A -85,B 0,C 180,E1 -7607.44,E2 -7607.44} C_VEL
LIN {X 0,Y 467.562,Z 362.24,A -85,B 0,C 180,E1 -7610.853,E2 -7610.853} C_VEL
LIN {X 0,Y 467.562,Z 362.244,A -85,B 0,C 180,E1 -7614.261,E2 -7614.261} C_VEL
LIN {X 0,Y 467.635,Z 362.402,A -85,B 0,C 180,E1 -7617.053,E2 -7617.053} C_VEL
LIN {X 0,Y 470.05,Z 373.645,A -85,B 0,C 180,E1 -7619.825,E2 -7619.825} C_VEL
LIN {X 0,Y 471.144,Z 379.66,A -85,B 0,C 180,E1 -7621.245,E2 -7621.245} C_VEL
LIN {X 0,Y 470.198,Z 393.829,A -85,B 0,C 180,E1 -7624.313,E2 -7624.313} C_VEL
LIN {X 0,Y 469.225,Z 409.177,A -85,B 0,C 180,E1 -7627.546,E2 -7627.546} C_VEL
LIN {X 0,Y 468.442,Z 424.631,A -85,B 0,C 180,E1 -7630.727,E2 -7630.727} C_VEL
LIN {X 0,Y 467.836,Z 439.837,A -85,B 0,C 180,E1 -7633.799,E2 -7633.799} C_VEL
LIN {X 0,Y 467.65,Z 445.58,A -85,B 0,C 180,E1 -7634.947,E2 -7634.947} C_VEL
LIN {X 0,Y 469.158,Z 459.838,A -85,B 0,C 180,E1 -7635.33,E2 -7635.33} C_VEL
LIN {X 0,Y 469.421,Z 464.051,A -85,B 0,C 180,E1 -7635.477,E2 -7635.477} C_VEL
LIN {X 0,Y 469.139,Z 476.848,A -85,B 0,C 180,E1 -7636.021,E2 -7636.021} C_VEL
LIN {X 0,Y 468.752,Z 488.217,A -85,B 0,C 180,E1 -7636.672,E2 -7636.672} C_VEL
LIN {X 0,Y 468.396,Z 499.04,A -85,B 0,C 180,E1 -7637.47,E2 -7637.47} C_VEL
LIN {X 0,Y 467.866,Z 510.415,A -85,B 0,C 180,E1 -7638.52,E2 -7638.52} C_VEL
LIN {X 0,Y 467.478,Z 519.826,A -85,B 0,C 180,E1 -7639.607,E2 -7639.607} C_VEL
LIN {X 0,Y 467.177,Z 528.909,A -85,B 0,C 180,E1 -7640.912,E2 -7640.912} C_VEL
LIN {X 0,Y 466.963,Z 536.195,A -85,B 0,C 180,E1 -7642.215,E2 -7642.215} C_VEL
LIN {X 0,Y 466.827,Z 542.001,A -85,B 0,C 180,E1 -7643.526,E2 -7643.526} C_VEL
LIN {X 0,Y 466.789,Z 546.483,A -85,B 0,C 180,E1 -7644.817,E2 -7644.817} C_VEL
LIN {X 0,Y 466.776,Z 548.85,A -85,B 0,C 180,E1 -7645.683,E2 -7645.683} C_VEL
LIN {X 0,Y 466.817,Z 550.778,A -85,B 0,C 180,E1 -7646.548,E2 -7646.548} C_VEL
LIN {X 0,Y 466.818,Z 552.239,A -85,B 0,C 180,E1 -7647.411,E2 -7647.411} C_VEL
LIN {X 0,Y 466.669,Z 553.849,A -85,B 0,C 180,E1 -7649.137,E2 -7649.137} C_VEL
LIN {X 0,Y 466.673,Z 554.054,A -85,B 0,C 180,E1 -7650,E2 -7650} C_VEL
LIN {X 0,Y 466.673,Z 553.806,A -85,B 0,C 180,E1 -7650.863,E2 -7650.863} C_VEL
LIN {X 0,Y 466.82,Z 552.101,A -85,B 0,C 180,E1 -7652.589,E2 -7652.589} C_VEL
LIN {X 0,Y 466.831,Z 550.602,A -85,B 0,C 180,E1 -7653.452,E2 -7653.452} C_VEL
LIN {X 0,Y 466.742,Z 547.481,A -85,B 0,C 180,E1 -7654.751,E2 -7654.751} C_VEL
LIN {X 0,Y 466.835,Z 543.27,A -85,B 0,C 180,E1 -7656.049,E2 -7656.049} C_VEL
LIN {X 0,Y 466.949,Z 536.791,A -85,B 0,C 180,E1 -7657.568,E2 -7657.568} C_VEL
LIN {X 0,Y 467.112,Z 529.721,A -85,B 0,C 180,E1 -7658.872,E2 -7658.872} C_VEL
LIN {X 0,Y 467.412,Z 520.842,A -85,B 0,C 180,E1 -7660.176,E2 -7660.176} C_VEL
LIN {X 0,Y 467.789,Z 510.72,A -85,B 0,C 180,E1 -7661.373,E2 -7661.373} C_VEL
LIN {X 0,Y 468.212,Z 499.858,A -85,B 0,C 180,E1 -7662.394,E2 -7662.394} C_VEL
LIN {X 0,Y 468.651,Z 488.868,A -85,B 0,C 180,E1 -7663.22,E2 -7663.22} C_VEL
LIN {X 0,Y 469.043,Z 476.898,A -85,B 0,C 180,E1 -7663.927,E2 -7663.927} C_VEL
LIN {X 0,Y 469.449,Z 463.646,A -85,B 0,C 180,E1 -7664.495,E2 -7664.495} C_VEL
LIN {X 0,Y 468.206,Z 450.781,A -85,B 0,C 180,E1 -7664.909,E2 -7664.909} C_VEL
LIN {X 0,Y 467.631,Z 444.915,A -85,B 0,C 180,E1 -7665.054,E2 -7665.054} C_VEL
LIN {X 0,Y 468.173,Z 428.26,A -85,B 0,C 180,E1 -7668.376,E2 -7668.376} C_VEL
LIN {X 0,Y 468.799,Z 415.167,A -85,B 0,C 180,E1 -7671.088,E2 -7671.088} C_VEL
LIN {X 0,Y 469.804,Z 400.085,A -85,B 0,C 180,E1 -7674.368,E2 -7674.368} C_VEL
LIN {X 0,Y 471.132,Z 386.635,A -85,B 0,C 180,E1 -7677.545,E2 -7677.545} C_VEL
LIN {X 0,Y 471.581,Z 381.062,A -85,B 0,C 180,E1 -7678.97,E2 -7678.97} C_VEL
LIN {X 0,Y 470.761,Z 375.856,A -85,B 0,C 180,E1 -7680.503,E2 -7680.503} C_VEL
LIN {X 0,Y 469.126,Z 368.581,A -85,B 0,C 180,E1 -7682.972,E2 -7682.972} C_VEL
LIN {X 0,Y 467.61,Z 362.377,A -85,B 0,C 180,E1 -7685.545,E2 -7685.545} C_VEL
LIN {X 0,Y 467.584,Z 362.243,A -85,B 0,C 180,E1 -7689.145,E2 -7689.145} C_VEL
LIN {X 0,Y 467.589,Z 362.243,A -85,B 0,C 180,E1 -7692.567,E2 -7692.567} C_VEL
LIN {X 0,Y 467.574,Z 362.245,A -85,B 0,C 180,E1 -7695.053,E2 -7695.053} C_VEL
LIN {X 0,Y 467.591,Z 362.241,A -85,B 0,C 180,E1 -7697.44,E2 -7697.44} C_VEL
LIN {X 0,Y 467.621,Z 362.239,A -85,B 0,C 180,E1 -7700.859,E2 -7700.859} C_VEL
LIN {X 0,Y 467.565,Z 362.246,A -85,B 0,C 180,E1 -7704.261,E2 -7704.261} C_VEL
LIN {X 0,Y 467.635,Z 362.42,A -85,B 0,C 180,E1 -7706.345,E2 -7706.345} C_VEL
LIN {X 0,Y 468.259,Z 366.271,A -85,B 0,C 180,E1 -7708.816,E2 -7708.816} C_VEL
LIN {X 0,Y 468.407,Z 369.129,A -85,B 0,C 180,E1 -7710.486,E2 -7710.486} C_VEL
LIN {X 0,Y 468.177,Z 374.082,A -85,B 0,C 180,E1 -7713.234,E2 -7713.234} C_VEL
LIN {X 0,Y 467.894,Z 379.979,A -85,B 0,C 180,E1 -7716.385,E2 -7716.385} C_VEL
LIN {X 0,Y 467.755,Z 384.723,A -85,B 0,C 180,E1 -7718.863,E2 -7718.863} C_VEL
LIN {X 0,Y 467.571,Z 390.059,A -85,B 0,C 180,E1 -7721.6,E2 -7721.6} C_VEL
LIN {X 0,Y 467.416,Z 395.436,A -85,B 0,C 180,E1 -7724.297,E2 -7724.297} C_VEL
LIN {X 0,Y 467.207,Z 402.749,A -85,B 0,C 180,E1 -7727.897,E2 -7727.897} C_VEL
LIN {X 0,Y 467.09,Z 408.294,A -85,B 0,C 180,E1 -7730.582,E2 -7730.582} C_VEL
LIN {X 0,Y 468.579,Z 416.992,A -85,B 0,C 180,E1 -7731.048,E2 -7731.048} C_VEL
LIN {X 0,Y 468.437,Z 425.667,A -85,B 0,C 180,E1 -7731.589,E2 -7731.589} C_VEL
LIN {X 0,Y 468.171,Z 434.77,A -85,B 0,C 180,E1 -7732.34,E2 -7732.34} C_VEL
LIN {X 0,Y 467.894,Z 441.918,A -85,B 0,C 180,E1 -7733.098,E2 -7733.098} C_VEL
LIN {X 0,Y 467.599,Z 448.343,A -85,B 0,C 180,E1 -7733.961,E2 -7733.961} C_VEL
LIN {X 0,Y 467.397,Z 454.539,A -85,B 0,C 180,E1 -7735.04,E2 -7735.04} C_VEL
LIN {X 0,Y 467.33,Z 459.131,A -85,B 0,C 180,E1 -7736.12,E2 -7736.12} C_VEL
LIN {X 0,Y 466.937,Z 462.97,A -85,B 0,C 180,E1 -7737.412,E2 -7737.412} C_VEL
LIN {X 0,Y 466.837,Z 464.588,A -85,B 0,C 180,E1 -7738.275,E2 -7738.275} C_VEL
LIN {X 0,Y 466.794,Z 465.515,A -85,B 0,C 180,E1 -7739.137,E2 -7739.137} C_VEL
LIN {X 0,Y 466.775,Z 465.773,A -85,B 0,C 180,E1 -7740,E2 -7740} C_VEL
LIN {X 0,Y 466.77,Z 465.367,A -85,B 0,C 180,E1 -7740.863,E2 -7740.863} C_VEL
LIN {X 0,Y 466.793,Z 464.29,A -85,B 0,C 180,E1 -7741.726,E2 -7741.726} C_VEL
LIN {X 0,Y 467.104,Z 461.345,A -85,B 0,C 180,E1 -7743.019,E2 -7743.019} C_VEL
LIN {X 0,Y 467.279,Z 456.661,A -85,B 0,C 180,E1 -7744.313,E2 -7744.313} C_VEL
LIN {X 0,Y 467.399,Z 451.198,A -85,B 0,C 180,E1 -7745.393,E2 -7745.393} C_VEL
LIN {X 0,Y 467.511,Z 445.544,A -85,B 0,C 180,E1 -7746.257,E2 -7746.257} C_VEL
LIN {X 0,Y 467.623,Z 439.002,A -85,B 0,C 180,E1 -7747.053,E2 -7747.053} C_VEL
LIN {X 0,Y 467.891,Z 430.301,A -85,B 0,C 180,E1 -7747.878,E2 -7747.878} C_VEL
LIN {X 0,Y 468.158,Z 421.276,A -85,B 0,C 180,E1 -7748.525,E2 -7748.525} C_VEL
LIN {X 0,Y 468.044,Z 414.47,A -85,B 0,C 180,E1 -7748.908,E2 -7748.908} C_VEL
LIN {X 0,Y 466.85,Z 406.459,A -85,B 0,C 180,E1 -7749.286,E2 -7749.286} C_VEL
LIN {X 0,Y 466.937,Z 400.227,A -85,B 0,C 180,E1 -7752.165,E2 -7752.165} C_VEL
LIN {X 0,Y 467.076,Z 392.634,A -85,B 0,C 180,E1 -7755.715,E2 -7755.715} C_VEL
LIN {X 0,Y 467.189,Z 385.022,A -85,B 0,C 180,E1 -7759.327,E2 -7759.327} C_VEL
LIN {X 0,Y 467.269,Z 379.299,A -85,B 0,C 180,E1 -7762.087,E2 -7762.087} C_VEL
LIN {X 0,Y 467.409,Z 373.498,A -85,B 0,C 180,E1 -7764.899,E2 -7764.899} C_VEL
LIN {X 0,Y 467.565,Z 367.654,A -85,B 0,C 180,E1 -7767.773,E2 -7767.773} C_VEL
LIN {X 0,Y 467.721,Z 362.226,A -85,B 0,C 180,E1 -7770.535,E2 -7770.535} C_VEL
LIN {X 0,Y 467.593,Z 362.239,A -85,B 0,C 180,E1 -7774.243,E2 -7774.243} C_VEL
LIN {X 0,Y 467.554,Z 362.244,A -85,B 0,C 180,E1 -7777.187,E2 -7777.187} C_VEL
LIN {X 0,Y 467.581,Z 362.241,A -85,B 0,C 180,E1 -7780.265,E2 -7780.265} C_VEL
LIN {X 0,Y 467.59,Z 362.24,A -85,B 0,C 180,E1 -7782.567,E2 -7782.567} C_VEL
LIN {X 0,Y 467.574,Z 362.242,A -85,B 0,C 180,E1 -7785.053,E2 -7785.053} C_VEL
LIN {X 0,Y 467.592,Z 362.24,A -85,B 0,C 180,E1 -7787.44,E2 -7787.44} C_VEL
LIN {X 0,Y 467.586,Z 362.242,A -85,B 0,C 180,E1 -7790.855,E2 -7790.855} C_VEL
LIN {X 0,Y 467.563,Z 362.243,A -85,B 0,C 180,E1 -7794.261,E2 -7794.261} C_VEL
LIN {X 0,Y 467.586,Z 362.24,A -85,B 0,C 180,E1 -7797.321,E2 -7797.321} C_VEL
LIN {X 0,Y 467.574,Z 362.242,A -85,B 0,C 180,E1 -7800.667,E2 -7800.667} C_VEL
LIN {X 0,Y 467.617,Z 362.237,A -85,B 0,C 180,E1 -7803.2,E2 -7803.2} C_VEL
LIN {X 0,Y 467.594,Z 362.241,A -85,B 0,C 180,E1 -7806.469,E2 -7806.469} C_VEL
LIN {X 0,Y 467.627,Z 362.237,A -85,B 0,C 180,E1 -7809.777,E2 -7809.777} C_VEL
LIN {X 0,Y 467.611,Z 362.238,A -85,B 0,C 180,E1 -7812.507,E2 -7812.507} C_VEL
LIN {X 0,Y 467.621,Z 362.235,A -85,B 0,C 180,E1 -7814.589,E2 -7814.589} C_VEL
LIN {X 0,Y 466.93,Z 362.321,A -85,B 0,C 180,E1 -7815.308,E2 -7815.308} C_VEL
LIN {X 0,Y 464.071,Z 362.68,A -85,B 0,C 180,E1 -7816.476,E2 -7816.476} C_VEL
LIN {X 0,Y 461.682,Z 362.974,A -85,B 0,C 180,E1 -7817.417,E2 -7817.417} C_VEL
LIN {X 0,Y 460.677,Z 363.104,A -85,B 0,C 180,E1 -7818.144,E2 -7818.144} C_VEL
LIN {X 0,Y 460.606,Z 363.108,A -85,B 0,C 180,E1 -7818.39,E2 -7818.39} C_VEL
LIN {X 0,Y 460.632,Z 363.107,A -85,B 0,C 180,E1 -7821.224,E2 -7821.224} C_VEL
LIN {X 0,Y 460.706,Z 363.097,A -85,B 0,C 180,E1 -7823.87,E2 -7823.87} C_VEL
